(* IEC 61131-3 sources: Codesys_MELSEC_Comm_Sample/src/SLMP_Function, 39 files *)

(* ---- SOCKADDRESS_IN.st ---- *)
TYPE SOCKADDRESS_IN :

STRUCT
    sin_family : INT;
    sin_port   : UINT;
    sin_addr   : UDINT;
    sin_zero   : ARRAY[0..7] OF BYTE;
END_STRUCT
END_TYPE

(* ---- GVL_SlmpConfig.st ---- *)
VAR_GLOBAL CONSTANT
    // LITE preset (active)
    SLMP_MAX_WORD_POINTS : UINT := 120;
    SLMP_MAX_BIT_POINTS : UINT := 960;
    SLMP_MAX_WORD_INDEX : UINT := 119;
    SLMP_MAX_BIT_INDEX : UINT := 959;

    // Buffer sizes for LITE preset (active)
    SLMP_READ_RX_INDEX_MAX : UINT := 511;
    SLMP_WRITE_TX_INDEX_MAX : UINT := 1023;
    SLMP_LAST_RESPONSE_INDEX_MAX : UINT := 63;

    (*
    // FULL preset (commented out)
    SLMP_MAX_WORD_POINTS : UINT := 960;
    SLMP_MAX_BIT_POINTS : UINT := 7168;
    SLMP_MAX_WORD_INDEX : UINT := 959;
    SLMP_MAX_BIT_INDEX : UINT := 7167;

    // Buffer sizes for FULL preset (commented out)
    SLMP_READ_RX_INDEX_MAX : UINT := 4095;
    SLMP_WRITE_TX_INDEX_MAX : UINT := 4095;
    SLMP_LAST_RESPONSE_INDEX_MAX : UINT := 255;
    *)
END_VAR

(* ---- GVL_SlmpDeviceCode.st ---- *)
VAR_GLOBAL CONSTANT
    SLMP_DEV_SM: UINT := 16#0091;
    SLMP_DEV_SD: UINT := 16#00A9;

    SLMP_DEV_X: UINT := 16#009C;
    SLMP_DEV_Y: UINT := 16#009D;

    SLMP_DEV_M: UINT := 16#0090;
    SLMP_DEV_L: UINT := 16#0092;

    SLMP_DEV_F: UINT := 16#0093;
    SLMP_DEV_V: UINT := 16#0094;

    SLMP_DEV_B: UINT := 16#00A0;
    SLMP_DEV_D: UINT := 16#00A8;
    SLMP_DEV_W: UINT := 16#00B4;

    SLMP_DEV_TS: UINT := 16#00C1;
    SLMP_DEV_TC: UINT := 16#00C0;
    SLMP_DEV_TN: UINT := 16#00C2;

    SLMP_DEV_LTS: UINT := 16#0051;
    SLMP_DEV_LTC: UINT := 16#0050;
    SLMP_DEV_LTN: UINT := 16#0052;

    SLMP_DEV_STS: UINT := 16#00C7;
    SLMP_DEV_STC: UINT := 16#00C6;
    SLMP_DEV_STN: UINT := 16#00C8;

    SLMP_DEV_LSTS: UINT := 16#0059;
    SLMP_DEV_LSTC: UINT := 16#0058;
    SLMP_DEV_LSTN: UINT := 16#005A;

    SLMP_DEV_CS: UINT := 16#00C4;
    SLMP_DEV_CC: UINT := 16#00C3;
    SLMP_DEV_CN: UINT := 16#00C5;

    SLMP_DEV_LCS: UINT := 16#0055;
    SLMP_DEV_LCC: UINT := 16#0054;
    SLMP_DEV_LCN: UINT := 16#0056;

    SLMP_DEV_SB: UINT := 16#00A1;
    SLMP_DEV_SW: UINT := 16#00B5;

    SLMP_DEV_S: UINT := 16#0098;

    SLMP_DEV_DX: UINT := 16#00A2;
    SLMP_DEV_DY: UINT := 16#00A3;

    SLMP_DEV_Z: UINT := 16#00CC;
    SLMP_DEV_LZ: UINT := 16#0062;

    SLMP_DEV_R: UINT := 16#00AF;
    SLMP_DEV_ZR: UINT := 16#00B0;

    SLMP_DEV_RD: UINT := 16#002C;
END_VAR

(* ---- GVL_SlmpRuntime.st ---- *)
VAR_GLOBAL
    g_uiSlmpSerialCounter : UINT := 0;
    g_udServiceInstanceCounter : UDINT := 0;
    g_aLockOwner : ARRAY[0..7] OF UDINT := [0,0,0,0,0,0,0,0];
    g_aLockIp : ARRAY[0..7] OF STRING := ['','','','','','','',''];
    g_aLockPort : ARRAY[0..7] OF UINT := [0,0,0,0,0,0,0,0];
    g_aLockUseUdp : ARRAY[0..7] OF BOOL := [FALSE,FALSE,FALSE,FALSE,FALSE,FALSE,FALSE,FALSE];

    g_aSockHandle : ARRAY[0..7] OF RTS_IEC_HANDLE := [
        RTS_INVALID_HANDLE, RTS_INVALID_HANDLE, RTS_INVALID_HANDLE, RTS_INVALID_HANDLE,
        RTS_INVALID_HANDLE, RTS_INVALID_HANDLE, RTS_INVALID_HANDLE, RTS_INVALID_HANDLE
    ];
    g_aSockConnected : ARRAY[0..7] OF BOOL := [FALSE,FALSE,FALSE,FALSE,FALSE,FALSE,FALSE,FALSE];
    g_aSockIp : ARRAY[0..7] OF STRING := ['','','','','','','',''];
    g_aSockPort : ARRAY[0..7] OF UINT := [0,0,0,0,0,0,0,0];
    g_aSockUseUdp : ARRAY[0..7] OF BOOL := [FALSE,FALSE,FALSE,FALSE,FALSE,FALSE,FALSE,FALSE];

    g_aLastTx : ARRAY[0..SLMP_WRITE_TX_INDEX_MAX] OF BYTE := [0];
    g_uiLastTxLen : UINT := 0;
    g_iLastTxSockSlot : INT := -1;
END_VAR

(* ---- GVL_SlmpSubCommand.st ---- *)
VAR_GLOBAL CONSTANT
    SLMP_SUB_WORD  : UINT := 16#0000;
    SLMP_SUB_BIT   : UINT := 16#0001;
    SLMP_SUB_WORD2 : UINT := 16#0002;
    SLMP_SUB_BIT2  : UINT := 16#0003;
END_VAR

(* ---- GVL_SlmpSubCommandByDevice.st ---- *)
VAR_GLOBAL CONSTANT
    SLMP_SUB_DEF_SM   : UINT := SLMP_SUB_BIT;
    SLMP_SUB_DEF_SD   : UINT := SLMP_SUB_WORD;

    SLMP_SUB_DEF_X    : UINT := SLMP_SUB_BIT;
    SLMP_SUB_DEF_Y    : UINT := SLMP_SUB_BIT;
    SLMP_SUB_DEF_M    : UINT := SLMP_SUB_BIT;
    SLMP_SUB_DEF_L    : UINT := SLMP_SUB_BIT;
    SLMP_SUB_DEF_F    : UINT := SLMP_SUB_BIT;
    SLMP_SUB_DEF_V    : UINT := SLMP_SUB_BIT;
    SLMP_SUB_DEF_B    : UINT := SLMP_SUB_BIT;

    SLMP_SUB_DEF_D    : UINT := SLMP_SUB_WORD;
    SLMP_SUB_DEF_W    : UINT := SLMP_SUB_WORD;

    SLMP_SUB_DEF_TS   : UINT := SLMP_SUB_BIT;
    SLMP_SUB_DEF_TC   : UINT := SLMP_SUB_BIT;
    SLMP_SUB_DEF_TN   : UINT := SLMP_SUB_WORD;

    SLMP_SUB_DEF_LTS  : UINT := SLMP_SUB_BIT2;
    SLMP_SUB_DEF_LTC  : UINT := SLMP_SUB_BIT2;
    SLMP_SUB_DEF_LTN  : UINT := SLMP_SUB_WORD2;

    SLMP_SUB_DEF_STS  : UINT := SLMP_SUB_BIT;
    SLMP_SUB_DEF_STC  : UINT := SLMP_SUB_BIT;
    SLMP_SUB_DEF_STN  : UINT := SLMP_SUB_WORD;

    SLMP_SUB_DEF_LSTS : UINT := SLMP_SUB_BIT2;
    SLMP_SUB_DEF_LSTC : UINT := SLMP_SUB_BIT2;
    SLMP_SUB_DEF_LSTN : UINT := SLMP_SUB_WORD2;

    SLMP_SUB_DEF_CS   : UINT := SLMP_SUB_BIT;
    SLMP_SUB_DEF_CC   : UINT := SLMP_SUB_BIT;
    SLMP_SUB_DEF_CN   : UINT := SLMP_SUB_WORD;

    SLMP_SUB_DEF_LCS  : UINT := SLMP_SUB_BIT2;
    SLMP_SUB_DEF_LCC  : UINT := SLMP_SUB_BIT2;
    SLMP_SUB_DEF_LCN  : UINT := SLMP_SUB_WORD;

    SLMP_SUB_DEF_SB   : UINT := SLMP_SUB_BIT;
    SLMP_SUB_DEF_SW   : UINT := SLMP_SUB_WORD;

    SLMP_SUB_DEF_S    : UINT := SLMP_SUB_BIT;

    SLMP_SUB_DEF_DX   : UINT := SLMP_SUB_BIT;
    SLMP_SUB_DEF_DY   : UINT := SLMP_SUB_BIT;

    SLMP_SUB_DEF_Z    : UINT := SLMP_SUB_WORD;
    SLMP_SUB_DEF_LZ   : UINT := SLMP_SUB_WORD2;

    SLMP_SUB_DEF_R    : UINT := SLMP_SUB_WORD;
    SLMP_SUB_DEF_ZR   : UINT := SLMP_SUB_WORD;

    SLMP_SUB_DEF_RD   : UINT := SLMP_SUB_WORD2;

END_VAR

(* ---- F_SlmpAutoSubCommand.st ---- *)
FUNCTION F_SlmpAutoSubCommand : UINT
VAR_INPUT
    uiDeviceCode : UINT;
END_VAR

// === IMPLEMENTATION ===
CASE uiDeviceCode OF
    SLMP_DEV_D: F_SlmpAutoSubCommand := SLMP_SUB_DEF_D;
    SLMP_DEV_M: F_SlmpAutoSubCommand := SLMP_SUB_DEF_M;
    SLMP_DEV_X: F_SlmpAutoSubCommand := SLMP_SUB_DEF_X;
    SLMP_DEV_Y: F_SlmpAutoSubCommand := SLMP_SUB_DEF_Y;
    SLMP_DEV_L: F_SlmpAutoSubCommand := SLMP_SUB_DEF_L;
    SLMP_DEV_SM: F_SlmpAutoSubCommand := SLMP_SUB_DEF_SM;
    SLMP_DEV_SD: F_SlmpAutoSubCommand := SLMP_SUB_DEF_SD;
    SLMP_DEV_F: F_SlmpAutoSubCommand := SLMP_SUB_DEF_F;
    SLMP_DEV_V: F_SlmpAutoSubCommand := SLMP_SUB_DEF_V;
    SLMP_DEV_R: F_SlmpAutoSubCommand := SLMP_SUB_DEF_R;
    SLMP_DEV_W: F_SlmpAutoSubCommand := SLMP_SUB_DEF_W;
    SLMP_DEV_B: F_SlmpAutoSubCommand := SLMP_SUB_DEF_B;
    SLMP_DEV_TS: F_SlmpAutoSubCommand := SLMP_SUB_DEF_TS;
    SLMP_DEV_TC: F_SlmpAutoSubCommand := SLMP_SUB_DEF_TC;
    SLMP_DEV_TN: F_SlmpAutoSubCommand := SLMP_SUB_DEF_TN;
    SLMP_DEV_LTS: F_SlmpAutoSubCommand := SLMP_SUB_DEF_LTS;
    SLMP_DEV_LTC: F_SlmpAutoSubCommand := SLMP_SUB_DEF_LTC;
    SLMP_DEV_LTN: F_SlmpAutoSubCommand := SLMP_SUB_DEF_LTN;
    SLMP_DEV_STS: F_SlmpAutoSubCommand := SLMP_SUB_DEF_STS;
    SLMP_DEV_STC: F_SlmpAutoSubCommand := SLMP_SUB_DEF_STC;
    SLMP_DEV_STN: F_SlmpAutoSubCommand := SLMP_SUB_DEF_STN;
    SLMP_DEV_LSTS: F_SlmpAutoSubCommand := SLMP_SUB_DEF_LSTS;
    SLMP_DEV_LSTC: F_SlmpAutoSubCommand := SLMP_SUB_DEF_LSTC;
    SLMP_DEV_LSTN: F_SlmpAutoSubCommand := SLMP_SUB_DEF_LSTN;
    SLMP_DEV_CS: F_SlmpAutoSubCommand := SLMP_SUB_DEF_CS;
    SLMP_DEV_CC: F_SlmpAutoSubCommand := SLMP_SUB_DEF_CC;
    SLMP_DEV_CN: F_SlmpAutoSubCommand := SLMP_SUB_DEF_CN;
    SLMP_DEV_LCS: F_SlmpAutoSubCommand := SLMP_SUB_DEF_LCS;
    SLMP_DEV_LCC: F_SlmpAutoSubCommand := SLMP_SUB_DEF_LCC;
    SLMP_DEV_LCN: F_SlmpAutoSubCommand := SLMP_SUB_DEF_LCN;
    SLMP_DEV_SB: F_SlmpAutoSubCommand := SLMP_SUB_DEF_SB;
    SLMP_DEV_SW: F_SlmpAutoSubCommand := SLMP_SUB_DEF_SW;
    SLMP_DEV_ZR: F_SlmpAutoSubCommand := SLMP_SUB_DEF_ZR;
    SLMP_DEV_DX: F_SlmpAutoSubCommand := SLMP_SUB_DEF_DX;
    SLMP_DEV_DY: F_SlmpAutoSubCommand := SLMP_SUB_DEF_DY;
    SLMP_DEV_S: F_SlmpAutoSubCommand := SLMP_SUB_DEF_S;
    SLMP_DEV_Z: F_SlmpAutoSubCommand := SLMP_SUB_DEF_Z;
    SLMP_DEV_LZ: F_SlmpAutoSubCommand := SLMP_SUB_DEF_LZ;
    SLMP_DEV_RD: F_SlmpAutoSubCommand := SLMP_SUB_DEF_RD;
ELSE
    F_SlmpAutoSubCommand := SLMP_SUB_WORD;
END_CASE;

(* ---- F_SlmpClampPoints.st ---- *)
FUNCTION F_SlmpClampPoints : UINT
VAR_INPUT
    uiPoints : UINT;
    xBitMode : BOOL;
END_VAR

// === IMPLEMENTATION ===
IF uiPoints = 0 THEN
    F_SlmpClampPoints := 0;
ELSIF xBitMode THEN
    IF uiPoints > SLMP_MAX_BIT_POINTS THEN
        F_SlmpClampPoints := SLMP_MAX_BIT_POINTS;
    ELSE
        F_SlmpClampPoints := uiPoints;
    END_IF;
ELSE
    IF uiPoints > SLMP_MAX_WORD_POINTS THEN
        F_SlmpClampPoints := SLMP_MAX_WORD_POINTS;
    ELSE
        F_SlmpClampPoints := uiPoints;
    END_IF;
END_IF;

(* ---- F_SlmpEndCodeText.st ---- *)
FUNCTION F_SlmpEndCodeText : STRING
VAR_INPUT
    uiEndCode : UINT;
END_VAR

// === IMPLEMENTATION ===
CASE uiEndCode OF
    16#0000: F_SlmpEndCodeText := 'OK';
    16#0050: F_SlmpEndCodeText := 'OUT_OF_RANGE';
    16#C051: F_SlmpEndCodeText := 'POINTS_OR_HEAD_DEVICE_ERROR';
    16#C052: F_SlmpEndCodeText := 'COMMAND_NOT_SUPPORTED';
    16#C053: F_SlmpEndCodeText := 'SUBCOMMAND_NOT_SUPPORTED';
    16#C054: F_SlmpEndCodeText := 'DATA_FORMAT_ERROR';
    16#C055: F_SlmpEndCodeText := 'WRITE_PROTECTED';
    16#C056: F_SlmpEndCodeText := 'CPU_BUSY';
    16#C061: F_SlmpEndCodeText := 'REQUEST_DATA_LENGTH_ERROR';
    16#CE10: F_SlmpEndCodeText := 'NETWORK_PARAMETER_ERROR';
    16#CE11: F_SlmpEndCodeText := 'DESTINATION_PARAMETER_ERROR';
ELSE
    F_SlmpEndCodeText := 'UNKNOWN_END_CODE';
END_CASE;

(* ---- F_SlmpIsBitSubCommand.st ---- *)
FUNCTION F_SlmpIsBitSubCommand : BOOL
VAR_INPUT
    uiSubCommand : UINT;
END_VAR

// === IMPLEMENTATION ===
F_SlmpIsBitSubCommand := (uiSubCommand = SLMP_SUB_BIT) OR (uiSubCommand = SLMP_SUB_BIT2);

(* ---- F_SlmpNextSerialNo.st ---- *)
FUNCTION F_SlmpNextSerialNo : UINT
VAR_INPUT
    uiSeed : UINT := 1;
END_VAR

// === IMPLEMENTATION ===
IF g_uiSlmpSerialCounter = 0 THEN
    IF uiSeed = 0 THEN
        g_uiSlmpSerialCounter := 1;
    ELSE
        g_uiSlmpSerialCounter := uiSeed;
    END_IF;
ELSE
    g_uiSlmpSerialCounter := g_uiSlmpSerialCounter + 1;
    IF g_uiSlmpSerialCounter = 0 THEN
        g_uiSlmpSerialCounter := 1;
    END_IF;
END_IF;

F_SlmpNextSerialNo := g_uiSlmpSerialCounter;

(* ---- F_SlmpResolveSubCommand.st ---- *)
FUNCTION F_SlmpResolveSubCommand : UINT
VAR_INPUT
    uiDeviceCode    : UINT;
    xAutoSubCommand : BOOL;
    uiSubCommand    : UINT;
END_VAR

// === IMPLEMENTATION ===
IF xAutoSubCommand THEN
    F_SlmpResolveSubCommand := F_SlmpAutoSubCommand(uiDeviceCode := uiDeviceCode);
ELSE
    F_SlmpResolveSubCommand := uiSubCommand;
END_IF;

(* ---- FB_SlmpCloseConnection.st ---- *)
FUNCTION_BLOCK FB_SlmpCloseConnection
VAR_INPUT
    xExecute : BOOL;
END_VAR
VAR_OUTPUT
    xDone    : BOOL;
END_VAR
VAR
    xExecPrev : BOOL := FALSE;
    iSlot     : INT := 0;
END_VAR

// === IMPLEMENTATION ===
xDone := FALSE;

IF xExecute AND (NOT xExecPrev) THEN
    FOR iSlot := 0 TO 7 DO
        IF GVL_SlmpRuntime.g_aSockHandle[iSlot] <> RTS_INVALID_HANDLE THEN
            SysSockClose(GVL_SlmpRuntime.g_aSockHandle[iSlot]);
            GVL_SlmpRuntime.g_aSockHandle[iSlot] := RTS_INVALID_HANDLE;
        END_IF;
        GVL_SlmpRuntime.g_aSockConnected[iSlot] := FALSE;
        GVL_SlmpRuntime.g_aSockIp[iSlot] := '';
        GVL_SlmpRuntime.g_aSockPort[iSlot] := 0;
        GVL_SlmpRuntime.g_aSockUseUdp[iSlot] := FALSE;

        GVL_SlmpRuntime.g_aLockOwner[iSlot] := 0;
        GVL_SlmpRuntime.g_aLockIp[iSlot] := '';
        GVL_SlmpRuntime.g_aLockPort[iSlot] := 0;
        GVL_SlmpRuntime.g_aLockUseUdp[iSlot] := FALSE;
    END_FOR;
    xDone := TRUE;
END_IF;

xExecPrev := xExecute;

(* ---- FB_SlmpCore.st ---- *)
FUNCTION_BLOCK FB_SlmpCore
VAR_OUTPUT
    diLastError : DINT;
END_VAR
VAR
    iSockSlot      : INT := -1;
    res            : RTS_IEC_RESULT := 0;
    sa             : SOCKADDRESS_IN;
    ipAddr         : UDINT := 0;
    liRet          : LINT := 0;
END_VAR

(* ---- FB_SlmpReadBitDevice.st ---- *)
FUNCTION_BLOCK FB_SlmpReadBitDevice
VAR_INPUT
    xExecute         : BOOL;
    sIp              : STRING;
    uiPort           : UINT;
    udiHeadDevNo     : UDINT := 100;
    uiDeviceCode     : UINT := 16#0090; // M
    xAutoSubCommand  : BOOL := TRUE;
    uiSubCommand     : UINT := 16#0001;
    uiPoints         : UINT := 1;
    tTimeout         : TIME := T#2S;
    uiRetryMax       : UINT := 2;
    tReconnectDelay  : TIME := T#500MS;
    xUse4E           : BOOL := FALSE;
    xUseUdp          : BOOL := FALSE;
    uiSerialNo       : UINT := 0;
END_VAR
VAR_OUTPUT
    xBusy            : BOOL;
    xDone            : BOOL;
    xError           : BOOL;
    diError          : DINT;
    uiRetryCount     : UINT;
    uiReadBits       : UINT;
    uiValue0         : UINT;
    aBits            : ARRAY[0..SLMP_MAX_BIT_INDEX] OF BOOL;
    aLastResponse    : ARRAY[0..SLMP_LAST_RESPONSE_INDEX_MAX] OF BYTE;
    uiLastResponseLen: UINT;
    uiLastEndCode    : UINT;
END_VAR
VAR
    step             : INT := 0;
    xExecPrev        : BOOL := FALSE;

    fbCore           : FB_SlmpCore;

    tx               : ARRAY[0..31] OF BYTE;
    rx               : ARRAY[0..SLMP_READ_RX_INDEX_MAX] OF BYTE;
    txLen            : LINT := 0;
    rxLen            : LINT := 0;
    lenReq           : UINT := 0;
    endCode          : UINT := 0;

    uiPointsReq      : UINT := 0;
    uiPointsEff      : UINT := 0;
    uiSubCmdEff      : UINT := 0;
    iDataStart       : DINT := 11;
    iEndCodeStart    : DINT := 9;
    iNeedRxLen       : LINT := 0;
    uiRxSerialNo     : UINT := 0;
    uiCopyLen        : UINT := 0;
    iByteOffset      : DINT := 0;
    byData           : BYTE := 0;
    idx              : UINT := 0;

    xStateTimeout    : BOOL := FALSE;
    xRetryTiming     : BOOL := FALSE;
    fbTimeout        : TON;
    fbReconnect      : TON;
END_VAR

// === IMPLEMENTATION ===
IF (xExecute AND NOT xExecPrev) THEN
    xBusy := TRUE;
    xDone := FALSE;
    xError := FALSE;
    diError := 0;
    uiRetryCount := 0;
    uiReadBits := 0;
    uiValue0 := 0;
    uiLastResponseLen := 0;
    uiLastEndCode := 0;
    FOR idx := 0 TO SLMP_MAX_BIT_INDEX DO
        aBits[idx] := FALSE;
    END_FOR;
    FOR idx := 0 TO SLMP_LAST_RESPONSE_INDEX_MAX DO
        aLastResponse[idx] := 0;
    END_FOR;
    step := 10;
END_IF;
xExecPrev := xExecute;

xStateTimeout := (step = 20) OR (step = 40) OR (step = 50);
fbTimeout(IN := xStateTimeout, PT := tTimeout);
fbReconnect(IN := xRetryTiming, PT := tReconnectDelay);

IF (step <> 0) AND (step <> 80) AND fbTimeout.Q THEN
    diError := -1010;
    xError := TRUE;
    step := 90;
END_IF;

CASE step OF
    0:
        xRetryTiming := FALSE;

    10:
        uiSubCmdEff := F_SlmpResolveSubCommand(
            uiDeviceCode := uiDeviceCode,
            xAutoSubCommand := xAutoSubCommand,
            uiSubCommand := uiSubCommand
        );

        uiPointsReq := uiPoints;
        IF uiPointsReq = 0 THEN
            diError := -1000;
            xError := TRUE;
            xBusy := FALSE;
            step := 0;
        ELSE
            uiPointsEff := F_SlmpClampPoints(uiPoints := uiPointsReq, xBitMode := TRUE);
        END_IF;

        IF NOT xError THEN
            step := 20;
        END_IF;

    20:
        IF fbCore.OpenAndConnect(sIp := sIp, uiPort := uiPort, xUseUdp := xUseUdp) THEN
            step := 30;
        ELSE
            CASE fbCore.diLastError OF
                -1: diError := -1001;
                -2: diError := -1005;
                -3: diError := -1002;
            ELSE
                diError := -1002;
            END_CASE;
            xError := TRUE;
            step := 90;
        END_IF;

    30:
        lenReq := 12;
        IF xUse4E THEN
            iDataStart := 15;
            iEndCodeStart := 13;
            tx[0] := 16#54; tx[1] := 16#00;
            tx[2] := TO_BYTE(uiSerialNo AND 16#00FF);
            tx[3] := TO_BYTE(SHR(uiSerialNo, 8) AND 16#00FF);
            tx[4] := 16#00; tx[5] := 16#00;
            tx[6] := 16#00;
            tx[7] := 16#FF;
            tx[8] := 16#FF; tx[9] := 16#03;
            tx[10] := 16#00;
            tx[11] := TO_BYTE(lenReq AND 16#00FF);
            tx[12] := TO_BYTE(SHR(lenReq, 8) AND 16#00FF);
            tx[13] := 16#10; tx[14] := 16#00;
            tx[15] := 16#01; tx[16] := 16#04;
            tx[17] := TO_BYTE(uiSubCmdEff AND 16#00FF);
            tx[18] := TO_BYTE(SHR(uiSubCmdEff, 8) AND 16#00FF);
            tx[19] := TO_BYTE(udiHeadDevNo AND 16#000000FF);
            tx[20] := TO_BYTE(SHR(udiHeadDevNo, 8) AND 16#000000FF);
            tx[21] := TO_BYTE(SHR(udiHeadDevNo, 16) AND 16#000000FF);
            tx[22] := TO_BYTE(uiDeviceCode AND 16#00FF);
            tx[23] := TO_BYTE(uiPointsEff AND 16#00FF);
            tx[24] := TO_BYTE(SHR(uiPointsEff, 8) AND 16#00FF);
            txLen := 25;
        ELSE
            iDataStart := 11;
            iEndCodeStart := 9;
            tx[0] := 16#50; tx[1] := 16#00;
            tx[2] := 16#00;
            tx[3] := 16#FF;
            tx[4] := 16#FF; tx[5] := 16#03;
            tx[6] := 16#00;
            tx[7] := TO_BYTE(lenReq AND 16#00FF);
            tx[8] := TO_BYTE(SHR(lenReq, 8) AND 16#00FF);
            tx[9] := 16#10; tx[10] := 16#00;
            tx[11] := 16#01; tx[12] := 16#04;
            tx[13] := TO_BYTE(uiSubCmdEff AND 16#00FF);
            tx[14] := TO_BYTE(SHR(uiSubCmdEff, 8) AND 16#00FF);
            tx[15] := TO_BYTE(udiHeadDevNo AND 16#000000FF);
            tx[16] := TO_BYTE(SHR(udiHeadDevNo, 8) AND 16#000000FF);
            tx[17] := TO_BYTE(SHR(udiHeadDevNo, 16) AND 16#000000FF);
            tx[18] := TO_BYTE(uiDeviceCode AND 16#00FF);
            tx[19] := TO_BYTE(uiPointsEff AND 16#00FF);
            tx[20] := TO_BYTE(SHR(uiPointsEff, 8) AND 16#00FF);
            txLen := 21;
        END_IF;
        step := 40;

    40:
        IF NOT fbCore.SendBytes(pData := ADR(tx[0]), liLen := txLen) THEN
            diError := -1003;
            xError := TRUE;
            step := 90;
        ELSE
            step := 50;
        END_IF;

    50:
        rxLen := fbCore.RecvBytes(pData := ADR(rx[0]), liMaxLen := SIZEOF(rx));
        IF rxLen > 0 THEN
            uiCopyLen := 0;
            IF rxLen > TO_LINT(SLMP_LAST_RESPONSE_INDEX_MAX + 1) THEN
                uiCopyLen := SLMP_LAST_RESPONSE_INDEX_MAX + 1;
            ELSE
                uiCopyLen := TO_UINT(rxLen);
            END_IF;
            uiLastResponseLen := uiCopyLen;
            IF uiCopyLen > 0 THEN
                FOR idx := 0 TO (uiCopyLen - 1) DO
                    aLastResponse[idx] := rx[idx];
                END_FOR;
            END_IF;

            iNeedRxLen := iDataStart + TO_LINT((uiPointsEff + 1) / 2);
            IF rxLen < iNeedRxLen THEN
                diError := -1004;
                xError := TRUE;
                step := 90;
            ELSE
                IF xUse4E THEN
                    uiRxSerialNo := TO_UINT(rx[2]) OR SHL(TO_UINT(rx[3]), 8);
                    IF uiRxSerialNo <> uiSerialNo THEN
                        // Drop stale frame and keep waiting until timeout.
                        rxLen := 0;
                        uiLastResponseLen := 0;
                    END_IF;
                END_IF;
            END_IF;
            IF (NOT xError) AND (rxLen > 0) THEN
                endCode := TO_UINT(rx[iEndCodeStart]) OR SHL(TO_UINT(rx[iEndCodeStart + 1]), 8);
                uiLastEndCode := endCode;
                IF endCode <> 0 THEN
                    diError := TO_DINT(endCode);
                    xError := TRUE;
                    step := 90;
                ELSE
                    FOR idx := 0 TO (uiPointsEff - 1) DO
                        iByteOffset := iDataStart + TO_DINT(idx / 2);
                        byData := rx[iByteOffset];
                        IF (idx MOD 2) = 0 THEN
                            aBits[idx] := (byData AND 16#F0) <> 0;
                        ELSE
                            aBits[idx] := (byData AND 16#0F) <> 0;
                        END_IF;
                    END_FOR;
                    uiReadBits := uiPointsEff;
                    IF uiPointsEff > 0 THEN
                        IF aBits[0] THEN
                            uiValue0 := 1;
                        ELSE
                            uiValue0 := 0;
                        END_IF;
                    END_IF;
                    xDone := TRUE;
                    xBusy := FALSE;
                    step := 90;
                END_IF;
            END_IF;
        END_IF;

    80:
        xRetryTiming := TRUE;
        IF fbReconnect.Q THEN
            xRetryTiming := FALSE;
            step := 10;
        END_IF;

    90:
        IF xError THEN
            fbCore.CloseSocket();
        END_IF;

        IF xError AND (uiRetryCount < uiRetryMax) THEN
            uiRetryCount := uiRetryCount + 1;
            xError := FALSE;
            step := 80;
        ELSE
            xBusy := FALSE;
            step := 0;
        END_IF;
END_CASE;

(* ---- FB_SlmpReadBitService.st ---- *)
FUNCTION_BLOCK FB_SlmpReadBitService
VAR_INPUT
    xExecute        : BOOL;
    sIp             : STRING;
    uiPort          : UINT;
    udiHeadDevNo    : UDINT;
    uiDeviceCode    : UINT;
    uiPoints        : UINT;
    tTimeout        : TIME := T#2S;
    uiRetryMax      : UINT := 2;
    tReconnectDelay : TIME := T#500MS;
    xUse4E          : BOOL := FALSE;
    xUseUdp         : BOOL := FALSE;
    uiSerialNo      : UINT := 1;
END_VAR
VAR_OUTPUT
    xBusy           : BOOL;
    xDone           : BOOL;
    xError          : BOOL;
    diError         : DINT;
    uiRetryCount    : UINT;
    uiReadBits      : UINT;
    uiValue0        : UINT;
    aReadBits       : ARRAY[0..SLMP_MAX_BIT_INDEX] OF BOOL;
    aLastResponse   : ARRAY[0..SLMP_LAST_RESPONSE_INDEX_MAX] OF BYTE;
    uiLastResponseLen : UINT;
    uiLastEndCode   : UINT;
END_VAR
VAR
    fbReadBit       : FB_SlmpReadBitDevice;
    udInstanceId    : UDINT := 0;

    xExecPrev       : BOOL := FALSE;
    xPending        : BOOL := FALSE;
    xActive         : BOOL := FALSE;
    xExecPulse      : BOOL := FALSE;
    iLockIdx        : INT := -1;

    udiHeadLatched  : UDINT := 0;
    uiDeviceLatched : UINT := 0;
    uiPointsLatched : UINT := 0;
    uiSerialActive  : UINT := 0;

    idx             : UINT;
    uiSerialEff     : UINT;
    iSlot           : INT;
    iFreeSlot       : INT;
    xLocked         : BOOL;
END_VAR

// === IMPLEMENTATION ===
IF udInstanceId = 0 THEN
    GVL_SlmpRuntime.g_udServiceInstanceCounter := GVL_SlmpRuntime.g_udServiceInstanceCounter + 1;
    udInstanceId := GVL_SlmpRuntime.g_udServiceInstanceCounter;
    IF udInstanceId = 0 THEN
        udInstanceId := 1;
    END_IF;
END_IF;

IF xExecute AND (NOT xExecPrev) THEN
    IF (NOT xPending) AND (NOT xActive) THEN
        udiHeadLatched := udiHeadDevNo;
        uiDeviceLatched := uiDeviceCode;
        uiPointsLatched := uiPoints;
        xDone := FALSE;
        xError := FALSE;
        diError := 0;
        uiRetryCount := 0;
        xPending := TRUE;
    END_IF;
END_IF;
xExecPrev := xExecute;

xExecPulse := FALSE;
IF xPending AND (NOT xActive) THEN
    xLocked := FALSE;
    iFreeSlot := -1;
    FOR iSlot := 0 TO 7 DO
        IF (GVL_SlmpRuntime.g_aLockOwner[iSlot] <> 0) AND
           (GVL_SlmpRuntime.g_aLockIp[iSlot] = sIp) AND
           (GVL_SlmpRuntime.g_aLockPort[iSlot] = uiPort) AND
           (GVL_SlmpRuntime.g_aLockUseUdp[iSlot] = xUseUdp) THEN
            xLocked := TRUE;
            EXIT;
        END_IF;
        IF (iFreeSlot < 0) AND (GVL_SlmpRuntime.g_aLockOwner[iSlot] = 0) THEN
            iFreeSlot := iSlot;
        END_IF;
    END_FOR;

    IF (NOT xLocked) AND (iFreeSlot >= 0) THEN
        GVL_SlmpRuntime.g_aLockOwner[iFreeSlot] := udInstanceId;
        GVL_SlmpRuntime.g_aLockIp[iFreeSlot] := sIp;
        GVL_SlmpRuntime.g_aLockPort[iFreeSlot] := uiPort;
        GVL_SlmpRuntime.g_aLockUseUdp[iFreeSlot] := xUseUdp;
        iLockIdx := iFreeSlot;

        xActive := TRUE;
        xExecPulse := TRUE;
        IF xUse4E THEN
            uiSerialActive := F_SlmpNextSerialNo(uiSeed := uiSerialNo);
        END_IF;
    END_IF;
END_IF;

IF xActive THEN
    IF xUse4E THEN
        uiSerialEff := uiSerialActive;
        IF uiSerialEff = 0 THEN
            uiSerialEff := 1;
        END_IF;
    ELSE
        uiSerialEff := uiSerialNo;
    END_IF;

    fbReadBit(
        xExecute := xExecPulse,
        sIp := sIp,
        uiPort := uiPort,
        udiHeadDevNo := udiHeadLatched,
        uiDeviceCode := uiDeviceLatched,
        xAutoSubCommand := TRUE,
        uiSubCommand := 0,
        uiPoints := uiPointsLatched,
        tTimeout := tTimeout,
        uiRetryMax := uiRetryMax,
        tReconnectDelay := tReconnectDelay,
        xUse4E := xUse4E,
        xUseUdp := xUseUdp,
        uiSerialNo := uiSerialEff
    );
ELSE
    xBusy := xPending;
    IF NOT xExecute THEN
        xDone := FALSE;
        xError := FALSE;
        diError := 0;
        uiRetryCount := 0;
    END_IF;
    RETURN;
END_IF;

xBusy := fbReadBit.xBusy;
xDone := fbReadBit.xDone;
xError := fbReadBit.xError;
diError := fbReadBit.diError;
uiRetryCount := fbReadBit.uiRetryCount;

IF fbReadBit.xDone THEN
    uiReadBits := fbReadBit.uiReadBits;
    uiValue0 := fbReadBit.uiValue0;
    FOR idx := 0 TO SLMP_MAX_BIT_INDEX DO
        aReadBits[idx] := fbReadBit.aBits[idx];
    END_FOR;
    FOR idx := 0 TO SLMP_LAST_RESPONSE_INDEX_MAX DO
        aLastResponse[idx] := fbReadBit.aLastResponse[idx];
    END_FOR;
    uiLastResponseLen := fbReadBit.uiLastResponseLen;
    uiLastEndCode := fbReadBit.uiLastEndCode;
END_IF;

IF fbReadBit.xDone OR fbReadBit.xError THEN
    xPending := FALSE;
    xActive := FALSE;
    IF iLockIdx >= 0 THEN
        GVL_SlmpRuntime.g_aLockOwner[iLockIdx] := 0;
        GVL_SlmpRuntime.g_aLockIp[iLockIdx] := '';
        GVL_SlmpRuntime.g_aLockPort[iLockIdx] := 0;
        GVL_SlmpRuntime.g_aLockUseUdp[iLockIdx] := FALSE;
        iLockIdx := -1;
    END_IF;
END_IF;

(* ---- FB_SlmpReadDevice.st ---- *)
FUNCTION_BLOCK FB_SlmpReadDevice
VAR_INPUT
    xExecute         : BOOL;
    sIp              : STRING;
    uiPort           : UINT;
    udiHeadDevNo     : UDINT := 100;
    uiDeviceCode     : UINT := 16#00A8; // D
    xAutoSubCommand  : BOOL := TRUE;
    uiSubCommand     : UINT := 16#0000; // 0000: word, 0001: bit
    uiPoints         : UINT := 1;
    tTimeout         : TIME := T#2S;
    uiRetryMax       : UINT := 2;
    tReconnectDelay  : TIME := T#500MS;
    xUse4E           : BOOL := FALSE;
    uiSerialNo       : UINT := 0;
END_VAR
VAR_OUTPUT
    xBusy            : BOOL;
    xDone            : BOOL;
    xError           : BOOL;
    diError          : DINT;
    uiRetryCount     : UINT;
    uiReadWords      : UINT;
    uiReadBits       : UINT;
    uiValue0         : UINT;
    aValues          : ARRAY[0..SLMP_MAX_WORD_INDEX] OF UINT;
    aBits            : ARRAY[0..SLMP_MAX_BIT_INDEX] OF BOOL;
    aLastResponse    : ARRAY[0..SLMP_LAST_RESPONSE_INDEX_MAX] OF BYTE;
    uiLastResponseLen: UINT;
    uiLastEndCode    : UINT;
END_VAR
VAR
    step             : INT := 0;
    xExecPrev        : BOOL := FALSE;

    fbCore           : FB_SlmpCore;

    tx               : ARRAY[0..31] OF BYTE;
    rx               : ARRAY[0..SLMP_READ_RX_INDEX_MAX] OF BYTE;
    txLen            : LINT := 0;
    rxLen            : LINT := 0;
    lenReq           : UINT := 0;
    endCode          : UINT := 0;

    uiPointsReq      : UINT := 0;
    uiPointsEff      : UINT := 0;
    uiSubCmdEff      : UINT := 0;
    iDataStart       : DINT := 11;
    iEndCodeStart    : DINT := 9;
    iNeedRxLen       : LINT := 0;
    uiRxSerialNo     : UINT := 0;
    uiCopyLen        : UINT := 0;
    iByteOffset      : DINT := 0;
    byData           : BYTE := 0;
    idx              : UINT := 0;
    xBitMode         : BOOL := FALSE;

    xStateTimeout    : BOOL := FALSE;
    xRetryTiming     : BOOL := FALSE;
    fbTimeout        : TON;
    fbReconnect      : TON;
END_VAR

// === IMPLEMENTATION ===
IF (xExecute AND NOT xExecPrev) THEN
    xBusy := TRUE;
    xDone := FALSE;
    xError := FALSE;
    diError := 0;
    uiRetryCount := 0;
    uiReadWords := 0;
    uiReadBits := 0;
    uiValue0 := 0;
    uiLastResponseLen := 0;
    uiLastEndCode := 0;
    FOR idx := 0 TO SLMP_MAX_WORD_INDEX DO
        aValues[idx] := 0;
    END_FOR;
    FOR idx := 0 TO SLMP_MAX_BIT_INDEX DO
        aBits[idx] := FALSE;
    END_FOR;
    FOR idx := 0 TO SLMP_LAST_RESPONSE_INDEX_MAX DO
        aLastResponse[idx] := 0;
    END_FOR;
    step := 10;
END_IF;
xExecPrev := xExecute;

xStateTimeout := (step = 20) OR (step = 40) OR (step = 50);
fbTimeout(IN := xStateTimeout, PT := tTimeout);
fbReconnect(IN := xRetryTiming, PT := tReconnectDelay);

IF (step <> 0) AND (step <> 80) AND fbTimeout.Q THEN
    diError := -1010;
    xError := TRUE;
    step := 90;
END_IF;

CASE step OF
    0:
        xRetryTiming := FALSE;

    10:
        uiSubCmdEff := F_SlmpResolveSubCommand(
            uiDeviceCode := uiDeviceCode,
            xAutoSubCommand := xAutoSubCommand,
            uiSubCommand := uiSubCommand
        );
        xBitMode := F_SlmpIsBitSubCommand(uiSubCommand := uiSubCmdEff);

        uiPointsReq := uiPoints;
        IF uiPointsReq = 0 THEN
            diError := -1000;
            xError := TRUE;
            xBusy := FALSE;
            step := 0;
        ELSE
            uiPointsEff := F_SlmpClampPoints(uiPoints := uiPointsReq, xBitMode := xBitMode);
        END_IF;

        IF NOT xError THEN
            step := 20;
        END_IF;

    20:
        IF fbCore.OpenAndConnect(sIp := sIp, uiPort := uiPort) THEN
            step := 30;
        ELSE
            CASE fbCore.diLastError OF
                -1: diError := -1001;
                -2: diError := -1005;
                -3: diError := -1002;
            ELSE
                diError := -1002;
            END_CASE;
            xError := TRUE;
            step := 90;
        END_IF;

    30:
        lenReq := 12;
        IF xUse4E THEN
            iDataStart := 15;
            iEndCodeStart := 13;
            tx[0] := 16#54; tx[1] := 16#00;
            tx[2] := TO_BYTE(uiSerialNo AND 16#00FF);
            tx[3] := TO_BYTE(SHR(uiSerialNo, 8) AND 16#00FF);
            tx[4] := 16#00; tx[5] := 16#00;
            tx[6] := 16#00;
            tx[7] := 16#FF;
            tx[8] := 16#FF; tx[9] := 16#03;
            tx[10] := 16#00;
            tx[11] := TO_BYTE(lenReq AND 16#00FF);
            tx[12] := TO_BYTE(SHR(lenReq, 8) AND 16#00FF);
            tx[13] := 16#10; tx[14] := 16#00;
            tx[15] := 16#01; tx[16] := 16#04;
            tx[17] := TO_BYTE(uiSubCmdEff AND 16#00FF);
            tx[18] := TO_BYTE(SHR(uiSubCmdEff, 8) AND 16#00FF);
            tx[19] := TO_BYTE(udiHeadDevNo AND 16#000000FF);
            tx[20] := TO_BYTE(SHR(udiHeadDevNo, 8) AND 16#000000FF);
            tx[21] := TO_BYTE(SHR(udiHeadDevNo, 16) AND 16#000000FF);
            tx[22] := TO_BYTE(uiDeviceCode AND 16#00FF);
            tx[23] := TO_BYTE(uiPointsEff AND 16#00FF);
            tx[24] := TO_BYTE(SHR(uiPointsEff, 8) AND 16#00FF);
            txLen := 25;
        ELSE
            iDataStart := 11;
            iEndCodeStart := 9;
            tx[0] := 16#50; tx[1] := 16#00;
            tx[2] := 16#00;
            tx[3] := 16#FF;
            tx[4] := 16#FF; tx[5] := 16#03;
            tx[6] := 16#00;
            tx[7] := TO_BYTE(lenReq AND 16#00FF);
            tx[8] := TO_BYTE(SHR(lenReq, 8) AND 16#00FF);
            tx[9] := 16#10; tx[10] := 16#00;
            tx[11] := 16#01; tx[12] := 16#04;
            tx[13] := TO_BYTE(uiSubCmdEff AND 16#00FF);
            tx[14] := TO_BYTE(SHR(uiSubCmdEff, 8) AND 16#00FF);
            tx[15] := TO_BYTE(udiHeadDevNo AND 16#000000FF);
            tx[16] := TO_BYTE(SHR(udiHeadDevNo, 8) AND 16#000000FF);
            tx[17] := TO_BYTE(SHR(udiHeadDevNo, 16) AND 16#000000FF);
            tx[18] := TO_BYTE(uiDeviceCode AND 16#00FF);
            tx[19] := TO_BYTE(uiPointsEff AND 16#00FF);
            tx[20] := TO_BYTE(SHR(uiPointsEff, 8) AND 16#00FF);
            txLen := 21;
        END_IF;
        step := 40;

    40:
        IF NOT fbCore.SendBytes(pData := ADR(tx[0]), liLen := txLen) THEN
            diError := -1003;
            xError := TRUE;
            step := 90;
        ELSE
            step := 50;
        END_IF;

    50:
        rxLen := fbCore.RecvBytes(pData := ADR(rx[0]), liMaxLen := SIZEOF(rx));
        IF rxLen > 0 THEN
            uiCopyLen := 0;
            IF rxLen > TO_LINT(SLMP_LAST_RESPONSE_INDEX_MAX + 1) THEN
                uiCopyLen := SLMP_LAST_RESPONSE_INDEX_MAX + 1;
            ELSE
                uiCopyLen := TO_UINT(rxLen);
            END_IF;
            uiLastResponseLen := uiCopyLen;
            IF uiCopyLen > 0 THEN
                FOR idx := 0 TO (uiCopyLen - 1) DO
                    aLastResponse[idx] := rx[idx];
                END_FOR;
            END_IF;
            iNeedRxLen := CalcNeedRxLen();
            IF rxLen < iNeedRxLen THEN
                diError := -1004;
                xError := TRUE;
                step := 90;
            ELSE
                IF xUse4E THEN
                    uiRxSerialNo := TO_UINT(rx[2]) OR SHL(TO_UINT(rx[3]), 8);
                    IF uiRxSerialNo <> uiSerialNo THEN
                        // Drop stale frame and keep waiting until timeout.
                        rxLen := 0;
                        uiLastResponseLen := 0;
                    END_IF;
                END_IF;
            END_IF;
            IF (NOT xError) AND (rxLen > 0) THEN
                endCode := TO_UINT(rx[iEndCodeStart]) OR SHL(TO_UINT(rx[iEndCodeStart + 1]), 8);
                uiLastEndCode := endCode;
                IF endCode <> 0 THEN
                    diError := TO_DINT(endCode);
                    xError := TRUE;
                    step := 90;
                ELSE
                    DecodeReadData();
                    xDone := TRUE;
                    xBusy := FALSE;
                    step := 90;
                END_IF;
            END_IF;
        END_IF;

    80:
        xRetryTiming := TRUE;
        IF fbReconnect.Q THEN
            xRetryTiming := FALSE;
            step := 10;
        END_IF;

    90:
        IF xError THEN
            fbCore.CloseSocket();
        END_IF;

        IF xError AND (uiRetryCount < uiRetryMax) THEN
            uiRetryCount := uiRetryCount + 1;
            xError := FALSE;
            step := 80;
        ELSE
            xBusy := FALSE;
            step := 0;
        END_IF;
END_CASE;

(* ---- FB_SlmpReadDWordDevice.st ---- *)
FUNCTION_BLOCK FB_SlmpReadDWordDevice
VAR_INPUT
    xExecute         : BOOL;
    sIp              : STRING;
    uiPort           : UINT;
    udiHeadDevNo     : UDINT := 0;
    uiDeviceCode     : UINT := 16#00C2; // LTN
    uiPoints         : UINT := 1; // number of 2-word points
    tTimeout         : TIME := T#2S;
    uiRetryMax       : UINT := 2;
    tReconnectDelay  : TIME := T#500MS;
    xUse4E           : BOOL := FALSE;
    xUseUdp          : BOOL := FALSE;
    uiSerialNo       : UINT := 0;
END_VAR
VAR_OUTPUT
    xBusy            : BOOL;
    xDone            : BOOL;
    xError           : BOOL;
    diError          : DINT;
    uiRetryCount     : UINT;
    uiReadPoints     : UINT; // number of 2-word points
    udiValue0        : UDINT;
    aReadDWords      : ARRAY[0..SLMP_MAX_WORD_INDEX] OF UDINT;
    aLastResponse    : ARRAY[0..SLMP_LAST_RESPONSE_INDEX_MAX] OF BYTE;
    uiLastResponseLen: UINT;
    uiLastEndCode    : UINT;
END_VAR
VAR
    fbReadWord       : FB_SlmpReadWordDevice;
    uiPointsEff      : UINT := 0;
    idx              : UINT := 0;
    udiLow           : UDINT := 0;
    udiHigh          : UDINT := 0;
END_VAR

// === IMPLEMENTATION ===
uiPointsEff := uiPoints;
IF uiPointsEff > (SLMP_MAX_WORD_POINTS / 2) THEN
    uiPointsEff := SLMP_MAX_WORD_POINTS / 2;
END_IF;

fbReadWord(
    xExecute := xExecute,
    sIp := sIp,
    uiPort := uiPort,
    udiHeadDevNo := udiHeadDevNo,
    uiDeviceCode := uiDeviceCode,
    xAutoSubCommand := FALSE,
    uiSubCommand := SLMP_SUB_WORD2,
    uiPoints := uiPointsEff,
    tTimeout := tTimeout,
    uiRetryMax := uiRetryMax,
    tReconnectDelay := tReconnectDelay,
    xUse4E := xUse4E,
    xUseUdp := xUseUdp,
    uiSerialNo := uiSerialNo
);

xBusy := fbReadWord.xBusy;
xDone := fbReadWord.xDone;
xError := fbReadWord.xError;
diError := fbReadWord.diError;
uiRetryCount := fbReadWord.uiRetryCount;
uiLastResponseLen := fbReadWord.uiLastResponseLen;
uiLastEndCode := fbReadWord.uiLastEndCode;
FOR idx := 0 TO SLMP_LAST_RESPONSE_INDEX_MAX DO
    aLastResponse[idx] := fbReadWord.aLastResponse[idx];
END_FOR;

IF fbReadWord.xDone THEN
    uiReadPoints := uiPointsEff;
    FOR idx := 0 TO (uiPointsEff - 1) DO
        udiLow := TO_UDINT(fbReadWord.aValues[idx * 2]);
        udiHigh := TO_UDINT(fbReadWord.aValues[idx * 2 + 1]);
        aReadDWords[idx] := udiLow OR SHL(udiHigh, 16);
    END_FOR;
    IF uiPointsEff > 0 THEN
        udiValue0 := aReadDWords[0];
    END_IF;
END_IF;

(* ---- FB_SlmpReadPlcInfo.st ---- *)
FUNCTION_BLOCK FB_SlmpReadPlcInfo
VAR_INPUT
    xExecute         : BOOL;
    sIp              : STRING;
    uiPort           : UINT;
    tTimeout         : TIME := T#2S;
    uiRetryMax       : UINT := 2;
    tReconnectDelay  : TIME := T#500MS;
    xUse4E           : BOOL := FALSE;
    xUseUdp          : BOOL := FALSE;
    uiSerialNo       : UINT := 1;
END_VAR
VAR_OUTPUT
    xBusy            : BOOL;
    xDone            : BOOL;
    xError           : BOOL;
    diError          : DINT;
    uiRetryCount     : UINT;
    aCpuTypeNameRaw  : ARRAY[0..15] OF BYTE;
    uiCpuTypeCode    : UINT;
    xPlcRun          : BOOL;
    xPlcStop         : BOOL;
    uiPlcMode        : UINT; // 0: unknown, 1: run, 2: stop
    aLastResponse    : ARRAY[0..SLMP_LAST_RESPONSE_INDEX_MAX] OF BYTE;
    uiLastResponseLen: UINT;
    uiLastEndCode    : UINT;
    aLastResponseCpuInfo : ARRAY[0..SLMP_LAST_RESPONSE_INDEX_MAX] OF BYTE;
    uiLastResponseCpuInfoLen : UINT;
    uiLastEndCodeCpuInfo : UINT;
    aLastResponseSm403 : ARRAY[0..SLMP_LAST_RESPONSE_INDEX_MAX] OF BYTE;
    uiLastResponseSm403Len : UINT;
    uiLastEndCodeSm403 : UINT;
END_VAR
VAR
    step             : INT := 0;
    xExecPrev        : BOOL := FALSE;

    fbCore           : FB_SlmpCore;

    tx               : ARRAY[0..31] OF BYTE;
    rx               : ARRAY[0..SLMP_LAST_RESPONSE_INDEX_MAX] OF BYTE;
    txLen            : LINT := 0;
    rxLen            : LINT := 0;
    lenReq           : UINT := 0;
    endCode          : UINT := 0;
    byModeData       : BYTE := 0;

    iDataStart       : DINT := 11;
    iEndCodeStart    : DINT := 9;
    iNeedRxLen       : LINT := 0;
    idx              : UINT := 0;
    uiCopyLen        : UINT := 0;

    xStateTimeout    : BOOL := FALSE;
    xRetryTiming     : BOOL := FALSE;
    fbTimeout        : TON;
    fbReconnect      : TON;
END_VAR

// === IMPLEMENTATION ===
IF (xExecute AND NOT xExecPrev) THEN
    xBusy := TRUE;
    xDone := FALSE;
    xError := FALSE;
    diError := 0;
    uiRetryCount := 0;
    uiCpuTypeCode := 0;
    xPlcRun := FALSE;
    xPlcStop := FALSE;
    uiPlcMode := 0;
    uiLastResponseLen := 0;
    uiLastEndCode := 0;
    uiLastResponseCpuInfoLen := 0;
    uiLastEndCodeCpuInfo := 0;
    uiLastResponseSm403Len := 0;
    uiLastEndCodeSm403 := 0;
    FOR idx := 0 TO 15 DO
        aCpuTypeNameRaw[idx] := 0;
    END_FOR;
    FOR idx := 0 TO SLMP_LAST_RESPONSE_INDEX_MAX DO
        aLastResponse[idx] := 0;
        aLastResponseCpuInfo[idx] := 0;
        aLastResponseSm403[idx] := 0;
    END_FOR;
    step := 10;
END_IF;
xExecPrev := xExecute;

xStateTimeout := (step = 20) OR (step = 40) OR (step = 50) OR (step = 60) OR (step = 70);
fbTimeout(IN := xStateTimeout, PT := tTimeout);
fbReconnect(IN := xRetryTiming, PT := tReconnectDelay);

IF (step <> 0) AND (step <> 80) AND fbTimeout.Q THEN
    diError := -3010;
    xError := TRUE;
    step := 90;
END_IF;

CASE step OF
    0:
        xRetryTiming := FALSE;

    10:
        step := 20;

    20:
        IF fbCore.OpenAndConnect(sIp := sIp, uiPort := uiPort, xUseUdp := xUseUdp) THEN
            step := 30;
        ELSE
            CASE fbCore.diLastError OF
                -1: diError := -3001;
                -2: diError := -3005;
                -3: diError := -3002;
            ELSE
                diError := -3002;
            END_CASE;
            xError := TRUE;
            step := 90;
        END_IF;

    30:
        lenReq := 6; // monitor timer(2) + command(2) + subcommand(2)

        IF xUse4E THEN
            iDataStart := 15;
            iEndCodeStart := 13;
            tx[0] := 16#54; tx[1] := 16#00;
            tx[2] := TO_BYTE(uiSerialNo AND 16#00FF);
            tx[3] := TO_BYTE(SHR(uiSerialNo, 8) AND 16#00FF);
            tx[4] := 16#00; tx[5] := 16#00;
            tx[6] := 16#00;
            tx[7] := 16#FF;
            tx[8] := 16#FF; tx[9] := 16#03;
            tx[10] := 16#00;
            tx[11] := TO_BYTE(lenReq AND 16#00FF);
            tx[12] := TO_BYTE(SHR(lenReq, 8) AND 16#00FF);
            tx[13] := 16#10; tx[14] := 16#00;
            tx[15] := 16#01; tx[16] := 16#01;
            tx[17] := 16#00; tx[18] := 16#00;
            txLen := 19;
        ELSE
            iDataStart := 11;
            iEndCodeStart := 9;
            tx[0] := 16#50; tx[1] := 16#00;
            tx[2] := 16#00;
            tx[3] := 16#FF;
            tx[4] := 16#FF; tx[5] := 16#03;
            tx[6] := 16#00;
            tx[7] := TO_BYTE(lenReq AND 16#00FF);
            tx[8] := TO_BYTE(SHR(lenReq, 8) AND 16#00FF);
            tx[9] := 16#10; tx[10] := 16#00;
            tx[11] := 16#01; tx[12] := 16#01;
            tx[13] := 16#00; tx[14] := 16#00;
            txLen := 15;
        END_IF;

        step := 40;

    40:
        IF NOT fbCore.SendBytes(pData := ADR(tx[0]), liLen := txLen) THEN
            diError := -3003;
            xError := TRUE;
            step := 90;
        ELSE
            step := 50;
        END_IF;

    50:
        rxLen := fbCore.RecvBytes(pData := ADR(rx[0]), liMaxLen := SIZEOF(rx));
        IF rxLen > 0 THEN
            // Auto-detect response frame type from subheader.
            IF (rxLen >= 15) AND (rx[0] = 16#D4) AND (rx[1] = 16#00) THEN
                iDataStart := 15;
                iEndCodeStart := 13;
            ELSIF (rxLen >= 11) AND (rx[0] = 16#D0) AND (rx[1] = 16#00) THEN
                iDataStart := 11;
                iEndCodeStart := 9;
            END_IF;
            uiCopyLen := 0;
            IF rxLen > TO_LINT(SLMP_LAST_RESPONSE_INDEX_MAX + 1) THEN
                uiCopyLen := SLMP_LAST_RESPONSE_INDEX_MAX + 1;
            ELSE
                uiCopyLen := TO_UINT(rxLen);
            END_IF;
            uiLastResponseLen := uiCopyLen;
            uiLastResponseCpuInfoLen := uiCopyLen;
            IF uiCopyLen > 0 THEN
                FOR idx := 0 TO (uiCopyLen - 1) DO
                    aLastResponse[idx] := rx[idx];
                    aLastResponseCpuInfo[idx] := rx[idx];
                END_FOR;
            END_IF;
            iNeedRxLen := TO_LINT(iEndCodeStart) + 2;
            IF rxLen < iNeedRxLen THEN
                diError := -3004;
                xError := TRUE;
                step := 90;
            ELSE
                IF iEndCodeStart = 13 THEN
                    IF (TO_UINT(rx[2]) OR SHL(TO_UINT(rx[3]), 8)) <> uiSerialNo THEN
                        // Drop stale frame and keep waiting until timeout.
                        rxLen := 0;
                        uiLastResponseLen := 0;
                        uiLastResponseCpuInfoLen := 0;
                    END_IF;
                END_IF;
            END_IF;
            IF (NOT xError) AND (rxLen > 0) THEN
                endCode := TO_UINT(rx[iEndCodeStart]) OR SHL(TO_UINT(rx[iEndCodeStart + 1]), 8);
                uiLastEndCode := endCode;
                uiLastEndCodeCpuInfo := endCode;
                IF endCode <> 0 THEN
                    diError := TO_DINT(endCode);
                    xError := TRUE;
                    step := 90;
                ELSE
                    iNeedRxLen := TO_LINT(iDataStart) + 18; // 16-byte name + 2-byte code
                    IF rxLen < iNeedRxLen THEN
                        diError := -3004;
                        xError := TRUE;
                        step := 90;
                    ELSE
                        FOR idx := 0 TO 15 DO
                            aCpuTypeNameRaw[idx] := rx[iDataStart + TO_DINT(idx)];
                        END_FOR;
                        uiCpuTypeCode := TO_UINT(rx[iDataStart + 16]) OR SHL(TO_UINT(rx[iDataStart + 17]), 8);
                        step := 60;
                    END_IF;
                END_IF;
            END_IF;
        END_IF;

    60:
        lenReq := 12;
        IF xUse4E THEN
            iDataStart := 15;
            iEndCodeStart := 13;
            tx[0] := 16#54; tx[1] := 16#00;
            tx[2] := TO_BYTE(uiSerialNo AND 16#00FF);
            tx[3] := TO_BYTE(SHR(uiSerialNo, 8) AND 16#00FF);
            tx[4] := 16#00; tx[5] := 16#00;
            tx[6] := 16#00;
            tx[7] := 16#FF;
            tx[8] := 16#FF; tx[9] := 16#03;
            tx[10] := 16#00;
            tx[11] := TO_BYTE(lenReq AND 16#00FF);
            tx[12] := TO_BYTE(SHR(lenReq, 8) AND 16#00FF);
            tx[13] := 16#10; tx[14] := 16#00;
            tx[15] := 16#01; tx[16] := 16#04;
            tx[17] := 16#01; tx[18] := 16#00;
            tx[19] := TO_BYTE(403 AND 16#000000FF);
            tx[20] := TO_BYTE(SHR(403, 8) AND 16#000000FF);
            tx[21] := TO_BYTE(SHR(403, 16) AND 16#000000FF);
            tx[22] := TO_BYTE(SLMP_DEV_SM AND 16#00FF);
            tx[23] := 16#01;
            tx[24] := 16#00;
            txLen := 25;
        ELSE
            iDataStart := 11;
            iEndCodeStart := 9;
            tx[0] := 16#50; tx[1] := 16#00;
            tx[2] := 16#00;
            tx[3] := 16#FF;
            tx[4] := 16#FF; tx[5] := 16#03;
            tx[6] := 16#00;
            tx[7] := TO_BYTE(lenReq AND 16#00FF);
            tx[8] := TO_BYTE(SHR(lenReq, 8) AND 16#00FF);
            tx[9] := 16#10; tx[10] := 16#00;
            tx[11] := 16#01; tx[12] := 16#04;
            tx[13] := 16#01; tx[14] := 16#00;
            tx[15] := TO_BYTE(403 AND 16#000000FF);
            tx[16] := TO_BYTE(SHR(403, 8) AND 16#000000FF);
            tx[17] := TO_BYTE(SHR(403, 16) AND 16#000000FF);
            tx[18] := TO_BYTE(SLMP_DEV_SM AND 16#00FF);
            tx[19] := 16#01;
            tx[20] := 16#00;
            txLen := 21;
        END_IF;

        IF NOT fbCore.SendBytes(pData := ADR(tx[0]), liLen := txLen) THEN
            diError := -3003;
            xError := TRUE;
            step := 90;
        ELSE
            step := 70;
        END_IF;

    70:
        rxLen := fbCore.RecvBytes(pData := ADR(rx[0]), liMaxLen := SIZEOF(rx));
        IF rxLen > 0 THEN
            // Auto-detect response frame type from subheader.
            IF (rxLen >= 15) AND (rx[0] = 16#D4) AND (rx[1] = 16#00) THEN
                iDataStart := 15;
                iEndCodeStart := 13;
            ELSIF (rxLen >= 11) AND (rx[0] = 16#D0) AND (rx[1] = 16#00) THEN
                iDataStart := 11;
                iEndCodeStart := 9;
            END_IF;
            uiCopyLen := 0;
            IF rxLen > TO_LINT(SLMP_LAST_RESPONSE_INDEX_MAX + 1) THEN
                uiCopyLen := SLMP_LAST_RESPONSE_INDEX_MAX + 1;
            ELSE
                uiCopyLen := TO_UINT(rxLen);
            END_IF;
            uiLastResponseLen := uiCopyLen;
            uiLastResponseSm403Len := uiCopyLen;
            IF uiCopyLen > 0 THEN
                FOR idx := 0 TO (uiCopyLen - 1) DO
                    aLastResponse[idx] := rx[idx];
                    aLastResponseSm403[idx] := rx[idx];
                END_FOR;
            END_IF;
            iNeedRxLen := TO_LINT(iEndCodeStart) + 2;
            IF rxLen < iNeedRxLen THEN
                diError := -3004;
                xError := TRUE;
                step := 90;
            ELSE
                IF iEndCodeStart = 13 THEN
                    IF (TO_UINT(rx[2]) OR SHL(TO_UINT(rx[3]), 8)) <> uiSerialNo THEN
                        // Drop stale frame and keep waiting until timeout.
                        rxLen := 0;
                        uiLastResponseLen := 0;
                        uiLastResponseSm403Len := 0;
                    END_IF;
                END_IF;
            END_IF;
            IF (NOT xError) AND (rxLen > 0) THEN
                endCode := TO_UINT(rx[iEndCodeStart]) OR SHL(TO_UINT(rx[iEndCodeStart + 1]), 8);
                uiLastEndCode := endCode;
                uiLastEndCodeSm403 := endCode;
                IF endCode <> 0 THEN
                    diError := TO_DINT(endCode);
                    xError := TRUE;
                    step := 90;
                ELSE
                    iNeedRxLen := TO_LINT(iDataStart) + 1;
                    IF rxLen < iNeedRxLen THEN
                        diError := -3004;
                        xError := TRUE;
                        step := 90;
                    ELSE
                        byModeData := rx[iDataStart];
                        xPlcRun := (byModeData AND 16#F0) <> 0;
                        xPlcStop := NOT xPlcRun;
                        IF xPlcRun THEN
                            uiPlcMode := 1;
                        ELSE
                            uiPlcMode := 2;
                        END_IF;
                        xDone := TRUE;
                        xBusy := FALSE;
                        step := 90;
                    END_IF;
                END_IF;
            END_IF;
        END_IF;

    80:
        xRetryTiming := TRUE;
        IF fbReconnect.Q THEN
            xRetryTiming := FALSE;
            step := 10;
        END_IF;

    90:
        IF xError THEN
            fbCore.CloseSocket();
        END_IF;

        IF xError AND (uiRetryCount < uiRetryMax) THEN
            uiRetryCount := uiRetryCount + 1;
            xError := FALSE;
            step := 80;
        ELSE
            xBusy := FALSE;
            step := 0;
        END_IF;
END_CASE;

(* ---- FB_SlmpReadPlcInfoService.st ---- *)
FUNCTION_BLOCK FB_SlmpReadPlcInfoService
VAR_INPUT
    xExecute        : BOOL;
    sIp             : STRING;
    uiPort          : UINT;
    tTimeout        : TIME := T#2S;
    uiRetryMax      : UINT := 2;
    tReconnectDelay : TIME := T#500MS;
    xUse4E          : BOOL := FALSE;
    xUseUdp         : BOOL := FALSE;
    uiSerialNo      : UINT := 1;
END_VAR
VAR_OUTPUT
    xBusy           : BOOL;
    xDone           : BOOL;
    xError          : BOOL;
    diError         : DINT;
    uiRetryCount    : UINT;
    aPlcTypeNameRaw : ARRAY[0..15] OF BYTE;
    sPlcTypeName    : STRING(16);
    uiPlcTypeCode   : UINT;
    xPlcRun         : BOOL;
    xPlcStop        : BOOL;
    uiPlcMode       : UINT;
    aLastResponse   : ARRAY[0..SLMP_LAST_RESPONSE_INDEX_MAX] OF BYTE;
    uiLastResponseLen : UINT;
    uiLastEndCode   : UINT;
END_VAR
VAR
    fbReadPlcInfo   : FB_SlmpReadPlcInfo;
    udInstanceId    : UDINT := 0;

    xExecPrev       : BOOL := FALSE;
    xPending        : BOOL := FALSE;
    xActive         : BOOL := FALSE;
    xExecPulse      : BOOL := FALSE;
    iLockIdx        : INT := -1;
    uiSerialActive  : UINT := 0;

    idx             : UINT;
    uiSerialEff     : UINT;
    iSlot           : INT;
    iFreeSlot       : INT;
    xLocked         : BOOL;
    pTypeName       : POINTER TO BYTE;
    uiNameLen       : UINT;
END_VAR

// === IMPLEMENTATION ===
IF udInstanceId = 0 THEN
    GVL_SlmpRuntime.g_udServiceInstanceCounter := GVL_SlmpRuntime.g_udServiceInstanceCounter + 1;
    udInstanceId := GVL_SlmpRuntime.g_udServiceInstanceCounter;
    IF udInstanceId = 0 THEN
        udInstanceId := 1;
    END_IF;
END_IF;

IF xExecute AND (NOT xExecPrev) THEN
    IF (NOT xPending) AND (NOT xActive) THEN
        xDone := FALSE;
        xError := FALSE;
        diError := 0;
        uiRetryCount := 0;
        xPending := TRUE;
    END_IF;
END_IF;
xExecPrev := xExecute;

xExecPulse := FALSE;
IF xPending AND (NOT xActive) THEN
    xLocked := FALSE;
    iFreeSlot := -1;
    FOR iSlot := 0 TO 7 DO
        IF (GVL_SlmpRuntime.g_aLockOwner[iSlot] <> 0) AND
           (GVL_SlmpRuntime.g_aLockIp[iSlot] = sIp) AND
           (GVL_SlmpRuntime.g_aLockPort[iSlot] = uiPort) AND
           (GVL_SlmpRuntime.g_aLockUseUdp[iSlot] = xUseUdp) THEN
            xLocked := TRUE;
            EXIT;
        END_IF;
        IF (iFreeSlot < 0) AND (GVL_SlmpRuntime.g_aLockOwner[iSlot] = 0) THEN
            iFreeSlot := iSlot;
        END_IF;
    END_FOR;

    IF (NOT xLocked) AND (iFreeSlot >= 0) THEN
        GVL_SlmpRuntime.g_aLockOwner[iFreeSlot] := udInstanceId;
        GVL_SlmpRuntime.g_aLockIp[iFreeSlot] := sIp;
        GVL_SlmpRuntime.g_aLockPort[iFreeSlot] := uiPort;
        GVL_SlmpRuntime.g_aLockUseUdp[iFreeSlot] := xUseUdp;
        iLockIdx := iFreeSlot;

        xActive := TRUE;
        xExecPulse := TRUE;
        IF xUse4E THEN
            uiSerialActive := F_SlmpNextSerialNo(uiSeed := uiSerialNo);
        END_IF;
    END_IF;
END_IF;

IF xActive THEN
    IF xUse4E THEN
        uiSerialEff := uiSerialActive;
        IF uiSerialEff = 0 THEN
            uiSerialEff := 1;
        END_IF;
    ELSE
        uiSerialEff := uiSerialNo;
    END_IF;

    fbReadPlcInfo(
        xExecute := xExecPulse,
        sIp := sIp,
        uiPort := uiPort,
        tTimeout := tTimeout,
        uiRetryMax := uiRetryMax,
        tReconnectDelay := tReconnectDelay,
        xUse4E := xUse4E,
        xUseUdp := xUseUdp,
        uiSerialNo := uiSerialEff
    );
ELSE
    xBusy := xPending;
    IF NOT xExecute THEN
        xDone := FALSE;
        xError := FALSE;
        diError := 0;
        uiRetryCount := 0;
    END_IF;
    RETURN;
END_IF;

xBusy := fbReadPlcInfo.xBusy;
xDone := fbReadPlcInfo.xDone;
xError := fbReadPlcInfo.xError;
diError := fbReadPlcInfo.diError;
uiRetryCount := fbReadPlcInfo.uiRetryCount;

IF fbReadPlcInfo.xDone THEN
    FOR idx := 0 TO 15 DO
        aPlcTypeNameRaw[idx] := fbReadPlcInfo.aCpuTypeNameRaw[idx];
    END_FOR;

    pTypeName := ADR(sPlcTypeName);
    FOR idx := 0 TO 16 DO
        pTypeName[idx] := 0;
    END_FOR;
    uiNameLen := 0;
    FOR idx := 0 TO 15 DO
        IF aPlcTypeNameRaw[idx] = 0 THEN
            EXIT;
        END_IF;
        pTypeName[uiNameLen] := aPlcTypeNameRaw[idx];
        uiNameLen := uiNameLen + 1;
    END_FOR;
    pTypeName[uiNameLen] := 0;

    uiPlcTypeCode := fbReadPlcInfo.uiCpuTypeCode;
    xPlcRun := fbReadPlcInfo.xPlcRun;
    xPlcStop := fbReadPlcInfo.xPlcStop;
    uiPlcMode := fbReadPlcInfo.uiPlcMode;

    FOR idx := 0 TO SLMP_LAST_RESPONSE_INDEX_MAX DO
        aLastResponse[idx] := fbReadPlcInfo.aLastResponse[idx];
    END_FOR;
    uiLastResponseLen := fbReadPlcInfo.uiLastResponseLen;
    uiLastEndCode := fbReadPlcInfo.uiLastEndCode;
END_IF;

IF fbReadPlcInfo.xDone OR fbReadPlcInfo.xError THEN
    xPending := FALSE;
    xActive := FALSE;
    IF iLockIdx >= 0 THEN
        GVL_SlmpRuntime.g_aLockOwner[iLockIdx] := 0;
        GVL_SlmpRuntime.g_aLockIp[iLockIdx] := '';
        GVL_SlmpRuntime.g_aLockPort[iLockIdx] := 0;
        GVL_SlmpRuntime.g_aLockUseUdp[iLockIdx] := FALSE;
        iLockIdx := -1;
    END_IF;
END_IF;

(* ---- FB_SlmpReadWordDevice.st ---- *)
FUNCTION_BLOCK FB_SlmpReadWordDevice
VAR_INPUT
    xExecute         : BOOL;
    sIp              : STRING;
    uiPort           : UINT;
    udiHeadDevNo     : UDINT := 100;
    uiDeviceCode     : UINT := 16#00A8; // D
    xAutoSubCommand  : BOOL := TRUE;
    uiSubCommand     : UINT := 16#0000;
    uiPoints         : UINT := 1;
    tTimeout         : TIME := T#2S;
    uiRetryMax       : UINT := 2;
    tReconnectDelay  : TIME := T#500MS;
    xUse4E           : BOOL := FALSE;
    xUseUdp          : BOOL := FALSE;
    uiSerialNo       : UINT := 0;
END_VAR
VAR_OUTPUT
    xBusy            : BOOL;
    xDone            : BOOL;
    xError           : BOOL;
    diError          : DINT;
    uiRetryCount     : UINT;
    uiReadWords      : UINT;
    uiValue0         : UINT;
    aValues          : ARRAY[0..SLMP_MAX_WORD_INDEX] OF UINT;
    aLastResponse    : ARRAY[0..SLMP_LAST_RESPONSE_INDEX_MAX] OF BYTE;
    uiLastResponseLen: UINT;
    uiLastEndCode    : UINT;
END_VAR
VAR
    step             : INT := 0;
    xExecPrev        : BOOL := FALSE;

    fbCore           : FB_SlmpCore;

    tx               : ARRAY[0..31] OF BYTE;
    rx               : ARRAY[0..SLMP_READ_RX_INDEX_MAX] OF BYTE;
    txLen            : LINT := 0;
    rxLen            : LINT := 0;
    lenReq           : UINT := 0;
    endCode          : UINT := 0;

    uiPointsReq      : UINT := 0;
    uiPointsEff      : UINT := 0;
    uiPointsProto    : UINT := 0;
    uiSubCmdEff      : UINT := 0;
    xWord2Mode       : BOOL := FALSE;
    iDataStart       : DINT := 11;
    iEndCodeStart    : DINT := 9;
    iNeedRxLen       : LINT := 0;
    uiRxSerialNo     : UINT := 0;
    uiCopyLen        : UINT := 0;
    idx              : UINT := 0;

    xStateTimeout    : BOOL := FALSE;
    xRetryTiming     : BOOL := FALSE;
    fbTimeout        : TON;
    fbReconnect      : TON;
END_VAR

// === IMPLEMENTATION ===
IF (xExecute AND NOT xExecPrev) THEN
    xBusy := TRUE;
    xDone := FALSE;
    xError := FALSE;
    diError := 0;
    uiRetryCount := 0;
    uiReadWords := 0;
    uiValue0 := 0;
    uiLastResponseLen := 0;
    uiLastEndCode := 0;
    FOR idx := 0 TO SLMP_MAX_WORD_INDEX DO
        aValues[idx] := 0;
    END_FOR;
    FOR idx := 0 TO SLMP_LAST_RESPONSE_INDEX_MAX DO
        aLastResponse[idx] := 0;
    END_FOR;
    step := 10;
END_IF;
xExecPrev := xExecute;

xStateTimeout := (step = 20) OR (step = 40) OR (step = 50);
fbTimeout(IN := xStateTimeout, PT := tTimeout);
fbReconnect(IN := xRetryTiming, PT := tReconnectDelay);

IF (step <> 0) AND (step <> 80) AND fbTimeout.Q THEN
    diError := -1010;
    xError := TRUE;
    step := 90;
END_IF;

CASE step OF
    0:
        xRetryTiming := FALSE;

    10:
        uiSubCmdEff := F_SlmpResolveSubCommand(
            uiDeviceCode := uiDeviceCode,
            xAutoSubCommand := xAutoSubCommand,
            uiSubCommand := uiSubCommand
        );
        xWord2Mode := (uiSubCmdEff = SLMP_SUB_WORD2);

        uiPointsReq := uiPoints;
        IF uiPointsReq = 0 THEN
            diError := -1000;
            xError := TRUE;
            xBusy := FALSE;
            step := 0;
        ELSE
            uiPointsEff := F_SlmpClampPoints(uiPoints := uiPointsReq, xBitMode := FALSE);
            IF xWord2Mode THEN
                IF uiPointsEff > (SLMP_MAX_WORD_POINTS / 2) THEN
                    uiPointsEff := SLMP_MAX_WORD_POINTS / 2;
                END_IF;
                uiPointsProto := uiPointsEff * 2;
            ELSE
                uiPointsProto := uiPointsEff;
            END_IF;
        END_IF;

        IF NOT xError THEN
            step := 20;
        END_IF;

    20:
        IF fbCore.OpenAndConnect(sIp := sIp, uiPort := uiPort, xUseUdp := xUseUdp) THEN
            step := 30;
        ELSE
            CASE fbCore.diLastError OF
                -1: diError := -1001;
                -2: diError := -1005;
                -3: diError := -1002;
            ELSE
                diError := -1002;
            END_CASE;
            xError := TRUE;
            step := 90;
        END_IF;

    30:
        lenReq := 12;
        IF xUse4E THEN
            iDataStart := 15;
            iEndCodeStart := 13;
            tx[0] := 16#54; tx[1] := 16#00;
            tx[2] := TO_BYTE(uiSerialNo AND 16#00FF);
            tx[3] := TO_BYTE(SHR(uiSerialNo, 8) AND 16#00FF);
            tx[4] := 16#00; tx[5] := 16#00;
            tx[6] := 16#00;
            tx[7] := 16#FF;
            tx[8] := 16#FF; tx[9] := 16#03;
            tx[10] := 16#00;
            tx[11] := TO_BYTE(lenReq AND 16#00FF);
            tx[12] := TO_BYTE(SHR(lenReq, 8) AND 16#00FF);
            tx[13] := 16#10; tx[14] := 16#00;
            tx[15] := 16#01; tx[16] := 16#04;
            tx[17] := TO_BYTE(uiSubCmdEff AND 16#00FF);
            tx[18] := TO_BYTE(SHR(uiSubCmdEff, 8) AND 16#00FF);
            tx[19] := TO_BYTE(udiHeadDevNo AND 16#000000FF);
            tx[20] := TO_BYTE(SHR(udiHeadDevNo, 8) AND 16#000000FF);
            tx[21] := TO_BYTE(SHR(udiHeadDevNo, 16) AND 16#000000FF);
            tx[22] := TO_BYTE(uiDeviceCode AND 16#00FF);
            tx[23] := TO_BYTE(uiPointsProto AND 16#00FF);
            tx[24] := TO_BYTE(SHR(uiPointsProto, 8) AND 16#00FF);
            txLen := 25;
        ELSE
            iDataStart := 11;
            iEndCodeStart := 9;
            tx[0] := 16#50; tx[1] := 16#00;
            tx[2] := 16#00;
            tx[3] := 16#FF;
            tx[4] := 16#FF; tx[5] := 16#03;
            tx[6] := 16#00;
            tx[7] := TO_BYTE(lenReq AND 16#00FF);
            tx[8] := TO_BYTE(SHR(lenReq, 8) AND 16#00FF);
            tx[9] := 16#10; tx[10] := 16#00;
            tx[11] := 16#01; tx[12] := 16#04;
            tx[13] := TO_BYTE(uiSubCmdEff AND 16#00FF);
            tx[14] := TO_BYTE(SHR(uiSubCmdEff, 8) AND 16#00FF);
            tx[15] := TO_BYTE(udiHeadDevNo AND 16#000000FF);
            tx[16] := TO_BYTE(SHR(udiHeadDevNo, 8) AND 16#000000FF);
            tx[17] := TO_BYTE(SHR(udiHeadDevNo, 16) AND 16#000000FF);
            tx[18] := TO_BYTE(uiDeviceCode AND 16#00FF);
            tx[19] := TO_BYTE(uiPointsProto AND 16#00FF);
            tx[20] := TO_BYTE(SHR(uiPointsProto, 8) AND 16#00FF);
            txLen := 21;
        END_IF;
        step := 40;

    40:
        IF NOT fbCore.SendBytes(pData := ADR(tx[0]), liLen := txLen) THEN
            diError := -1003;
            xError := TRUE;
            step := 90;
        ELSE
            step := 50;
        END_IF;

    50:
        rxLen := fbCore.RecvBytes(pData := ADR(rx[0]), liMaxLen := SIZEOF(rx));
        IF rxLen > 0 THEN
            uiCopyLen := 0;
            IF rxLen > TO_LINT(SLMP_LAST_RESPONSE_INDEX_MAX + 1) THEN
                uiCopyLen := SLMP_LAST_RESPONSE_INDEX_MAX + 1;
            ELSE
                uiCopyLen := TO_UINT(rxLen);
            END_IF;
            uiLastResponseLen := uiCopyLen;
            IF uiCopyLen > 0 THEN
                FOR idx := 0 TO (uiCopyLen - 1) DO
                    aLastResponse[idx] := rx[idx];
                END_FOR;
            END_IF;

            IF xWord2Mode THEN
                iNeedRxLen := iDataStart + TO_LINT(uiPointsEff) * 4;
            ELSE
                iNeedRxLen := iDataStart + TO_LINT(uiPointsEff) * 2;
            END_IF;
            IF rxLen < iNeedRxLen THEN
                diError := -1004;
                xError := TRUE;
                step := 90;
            ELSE
                IF xUse4E THEN
                    uiRxSerialNo := TO_UINT(rx[2]) OR SHL(TO_UINT(rx[3]), 8);
                    IF uiRxSerialNo <> uiSerialNo THEN
                        // Drop stale frame and keep waiting until timeout.
                        rxLen := 0;
                        uiLastResponseLen := 0;
                    END_IF;
                END_IF;
            END_IF;
            IF (NOT xError) AND (rxLen > 0) THEN
                endCode := TO_UINT(rx[iEndCodeStart]) OR SHL(TO_UINT(rx[iEndCodeStart + 1]), 8);
                uiLastEndCode := endCode;
                IF endCode <> 0 THEN
                    diError := TO_DINT(endCode);
                    xError := TRUE;
                    step := 90;
                ELSE
                    IF xWord2Mode THEN
                        FOR idx := 0 TO (uiPointsEff - 1) DO
                            aValues[idx * 2] := TO_UINT(rx[iDataStart + TO_DINT(idx) * 4]) OR
                                SHL(TO_UINT(rx[iDataStart + TO_DINT(idx) * 4 + 1]), 8);
                            aValues[idx * 2 + 1] := TO_UINT(rx[iDataStart + TO_DINT(idx) * 4 + 2]) OR
                                SHL(TO_UINT(rx[iDataStart + TO_DINT(idx) * 4 + 3]), 8);
                        END_FOR;
                        uiReadWords := uiPointsEff * 2;
                    ELSE
                        FOR idx := 0 TO (uiPointsEff - 1) DO
                            aValues[idx] := TO_UINT(rx[iDataStart + TO_DINT(idx) * 2]) OR
                                SHL(TO_UINT(rx[iDataStart + TO_DINT(idx) * 2 + 1]), 8);
                        END_FOR;
                        uiReadWords := uiPointsEff;
                    END_IF;
                    uiValue0 := aValues[0];
                    xDone := TRUE;
                    xBusy := FALSE;
                    step := 90;
                END_IF;
            END_IF;
        END_IF;

    80:
        xRetryTiming := TRUE;
        IF fbReconnect.Q THEN
            xRetryTiming := FALSE;
            step := 10;
        END_IF;

    90:
        IF xError THEN
            fbCore.CloseSocket();
        END_IF;

        IF xError AND (uiRetryCount < uiRetryMax) THEN
            uiRetryCount := uiRetryCount + 1;
            xError := FALSE;
            step := 80;
        ELSE
            xBusy := FALSE;
            step := 0;
        END_IF;
END_CASE;

(* ---- FB_SlmpReadWordService.st ---- *)
FUNCTION_BLOCK FB_SlmpReadWordService
VAR_INPUT
    xExecute        : BOOL;
    sIp             : STRING;
    uiPort          : UINT;
    udiHeadDevNo    : UDINT;
    uiDeviceCode    : UINT;
    uiPoints        : UINT;
    tTimeout        : TIME := T#2S;
    uiRetryMax      : UINT := 2;
    tReconnectDelay : TIME := T#500MS;
    xUse4E          : BOOL := FALSE;
    xUseUdp         : BOOL := FALSE;
    uiSerialNo      : UINT := 1;
END_VAR
VAR_OUTPUT
    xBusy           : BOOL;
    xDone           : BOOL;
    xError          : BOOL;
    diError         : DINT;
    uiRetryCount    : UINT;
    uiReadWords     : UINT;
    uiValue0        : UINT;
    aReadValues     : ARRAY[0..SLMP_MAX_WORD_INDEX] OF UINT;
    aLastResponse   : ARRAY[0..SLMP_LAST_RESPONSE_INDEX_MAX] OF BYTE;
    uiLastResponseLen : UINT;
    uiLastEndCode   : UINT;
END_VAR
VAR
    fbReadWord      : FB_SlmpReadWordDevice;
    udInstanceId    : UDINT := 0;

    xExecPrev       : BOOL := FALSE;
    xPending        : BOOL := FALSE;
    xActive         : BOOL := FALSE;
    xExecPulse      : BOOL := FALSE;
    iLockIdx        : INT := -1;

    udiHeadLatched  : UDINT := 0;
    uiDeviceLatched : UINT := 0;
    uiPointsLatched : UINT := 0;
    uiSerialActive  : UINT := 0;

    idx             : UINT;
    uiSerialEff     : UINT;
    iSlot           : INT;
    iFreeSlot       : INT;
    xLocked         : BOOL;
END_VAR

// === IMPLEMENTATION ===
IF udInstanceId = 0 THEN
    GVL_SlmpRuntime.g_udServiceInstanceCounter := GVL_SlmpRuntime.g_udServiceInstanceCounter + 1;
    udInstanceId := GVL_SlmpRuntime.g_udServiceInstanceCounter;
    IF udInstanceId = 0 THEN
        udInstanceId := 1;
    END_IF;
END_IF;

IF xExecute AND (NOT xExecPrev) THEN
    IF (NOT xPending) AND (NOT xActive) THEN
        udiHeadLatched := udiHeadDevNo;
        uiDeviceLatched := uiDeviceCode;
        uiPointsLatched := uiPoints;
        xDone := FALSE;
        xError := FALSE;
        diError := 0;
        uiRetryCount := 0;
        xPending := TRUE;
    END_IF;
END_IF;
xExecPrev := xExecute;

xExecPulse := FALSE;
IF xPending AND (NOT xActive) THEN
    xLocked := FALSE;
    iFreeSlot := -1;
    FOR iSlot := 0 TO 7 DO
        IF (GVL_SlmpRuntime.g_aLockOwner[iSlot] <> 0) AND
           (GVL_SlmpRuntime.g_aLockIp[iSlot] = sIp) AND
           (GVL_SlmpRuntime.g_aLockPort[iSlot] = uiPort) AND
           (GVL_SlmpRuntime.g_aLockUseUdp[iSlot] = xUseUdp) THEN
            xLocked := TRUE;
            EXIT;
        END_IF;
        IF (iFreeSlot < 0) AND (GVL_SlmpRuntime.g_aLockOwner[iSlot] = 0) THEN
            iFreeSlot := iSlot;
        END_IF;
    END_FOR;

    IF (NOT xLocked) AND (iFreeSlot >= 0) THEN
        GVL_SlmpRuntime.g_aLockOwner[iFreeSlot] := udInstanceId;
        GVL_SlmpRuntime.g_aLockIp[iFreeSlot] := sIp;
        GVL_SlmpRuntime.g_aLockPort[iFreeSlot] := uiPort;
        GVL_SlmpRuntime.g_aLockUseUdp[iFreeSlot] := xUseUdp;
        iLockIdx := iFreeSlot;

        xActive := TRUE;
        xExecPulse := TRUE;
        IF xUse4E THEN
            uiSerialActive := F_SlmpNextSerialNo(uiSeed := uiSerialNo);
        END_IF;
    END_IF;
END_IF;

IF xActive THEN
    IF xUse4E THEN
        uiSerialEff := uiSerialActive;
        IF uiSerialEff = 0 THEN
            uiSerialEff := 1;
        END_IF;
    ELSE
        uiSerialEff := uiSerialNo;
    END_IF;

    fbReadWord(
        xExecute := xExecPulse,
        sIp := sIp,
        uiPort := uiPort,
        udiHeadDevNo := udiHeadLatched,
        uiDeviceCode := uiDeviceLatched,
        xAutoSubCommand := TRUE,
        uiSubCommand := 0,
        uiPoints := uiPointsLatched,
        tTimeout := tTimeout,
        uiRetryMax := uiRetryMax,
        tReconnectDelay := tReconnectDelay,
        xUse4E := xUse4E,
        xUseUdp := xUseUdp,
        uiSerialNo := uiSerialEff
    );
ELSE
    xBusy := xPending;
    IF NOT xExecute THEN
        xDone := FALSE;
        xError := FALSE;
        diError := 0;
        uiRetryCount := 0;
    END_IF;
    RETURN;
END_IF;

xBusy := fbReadWord.xBusy;
xDone := fbReadWord.xDone;
xError := fbReadWord.xError;
diError := fbReadWord.diError;
uiRetryCount := fbReadWord.uiRetryCount;

IF fbReadWord.xDone THEN
    uiReadWords := fbReadWord.uiReadWords;
    uiValue0 := fbReadWord.uiValue0;
    FOR idx := 0 TO SLMP_MAX_WORD_INDEX DO
        aReadValues[idx] := fbReadWord.aValues[idx];
    END_FOR;
    FOR idx := 0 TO SLMP_LAST_RESPONSE_INDEX_MAX DO
        aLastResponse[idx] := fbReadWord.aLastResponse[idx];
    END_FOR;
    uiLastResponseLen := fbReadWord.uiLastResponseLen;
    uiLastEndCode := fbReadWord.uiLastEndCode;
END_IF;

IF fbReadWord.xDone OR fbReadWord.xError THEN
    xPending := FALSE;
    xActive := FALSE;
    IF iLockIdx >= 0 THEN
        GVL_SlmpRuntime.g_aLockOwner[iLockIdx] := 0;
        GVL_SlmpRuntime.g_aLockIp[iLockIdx] := '';
        GVL_SlmpRuntime.g_aLockPort[iLockIdx] := 0;
        GVL_SlmpRuntime.g_aLockUseUdp[iLockIdx] := FALSE;
        iLockIdx := -1;
    END_IF;
END_IF;

(* ---- FB_SlmpWriteBitDevice.st ---- *)
FUNCTION_BLOCK FB_SlmpWriteBitDevice
VAR_INPUT
    xExecute         : BOOL;
    sIp              : STRING;
    uiPort           : UINT;
    udiHeadDevNo     : UDINT := 100;
    uiDeviceCode     : UINT := 16#0090; // M
    xAutoSubCommand  : BOOL := TRUE;
    uiSubCommand     : UINT := 16#0001;
    uiPoints         : UINT := 1;
    aWriteBits       : ARRAY[0..SLMP_MAX_BIT_INDEX] OF BOOL;
    tTimeout         : TIME := T#2S;
    uiRetryMax       : UINT := 2;
    tReconnectDelay  : TIME := T#500MS;
    xUse4E           : BOOL := FALSE;
    xUseUdp          : BOOL := FALSE;
    uiSerialNo       : UINT := 0;
END_VAR
VAR_OUTPUT
    xBusy            : BOOL;
    xDone            : BOOL;
    xError           : BOOL;
    diError          : DINT;
    uiRetryCount     : UINT;
    aLastResponse    : ARRAY[0..SLMP_LAST_RESPONSE_INDEX_MAX] OF BYTE;
    uiLastResponseLen: UINT;
    uiLastEndCode    : UINT;
END_VAR
VAR
    step             : INT := 0;
    xExecPrev        : BOOL := FALSE;

    fbCore           : FB_SlmpCore;

    tx               : ARRAY[0..SLMP_WRITE_TX_INDEX_MAX] OF BYTE;
    rx               : ARRAY[0..SLMP_LAST_RESPONSE_INDEX_MAX] OF BYTE;
    txLen            : LINT := 0;
    rxLen            : LINT := 0;
    lenReq           : UINT := 0;
    endCode          : UINT := 0;

    uiPointsReq      : UINT := 0;
    uiPointsEff      : UINT := 0;
    uiSubCmdEff      : UINT := 0;
    idx              : UINT := 0;
    iDataStart       : DINT := 21;
    iEndCodeStart    : DINT := 9;
    iMinRxLen        : LINT := 11;
    uiRxSerialNo     : UINT := 0;
    uiCopyLen        : UINT := 0;
    iPayloadBytes    : LINT := 0;
    iByteOffset      : DINT := 0;

    xStateTimeout    : BOOL := FALSE;
    xRetryTiming     : BOOL := FALSE;
    fbTimeout        : TON;
    fbReconnect      : TON;
END_VAR

// === IMPLEMENTATION ===
IF (xExecute AND NOT xExecPrev) THEN
    xBusy := TRUE;
    xDone := FALSE;
    xError := FALSE;
    diError := 0;
    uiRetryCount := 0;
    uiLastResponseLen := 0;
    uiLastEndCode := 0;
    FOR idx := 0 TO SLMP_LAST_RESPONSE_INDEX_MAX DO
        aLastResponse[idx] := 0;
    END_FOR;
    step := 10;
END_IF;
xExecPrev := xExecute;

xStateTimeout := (step = 20) OR (step = 40) OR (step = 50);
fbTimeout(IN := xStateTimeout, PT := tTimeout);
fbReconnect(IN := xRetryTiming, PT := tReconnectDelay);

IF (step <> 0) AND (step <> 80) AND fbTimeout.Q THEN
    diError := -2010;
    xError := TRUE;
    step := 90;
END_IF;

CASE step OF
    0:
        xRetryTiming := FALSE;

    10:
        uiSubCmdEff := F_SlmpResolveSubCommand(
            uiDeviceCode := uiDeviceCode,
            xAutoSubCommand := xAutoSubCommand,
            uiSubCommand := uiSubCommand
        );

        uiPointsReq := uiPoints;
        IF uiPointsReq = 0 THEN
            diError := -2000;
            xError := TRUE;
            xBusy := FALSE;
            step := 0;
        ELSE
            uiPointsEff := F_SlmpClampPoints(uiPoints := uiPointsReq, xBitMode := TRUE);
        END_IF;

        IF NOT xError THEN
            step := 20;
        END_IF;

    20:
        IF fbCore.OpenAndConnect(sIp := sIp, uiPort := uiPort, xUseUdp := xUseUdp) THEN
            step := 30;
        ELSE
            CASE fbCore.diLastError OF
                -1: diError := -2001;
                -2: diError := -2005;
                -3: diError := -2002;
            ELSE
                diError := -2002;
            END_CASE;
            xError := TRUE;
            step := 90;
        END_IF;

    30:
        IF xUse4E THEN
            iDataStart := 25;
            iEndCodeStart := 13;
            iMinRxLen := 15;
        ELSE
            iDataStart := 21;
            iEndCodeStart := 9;
            iMinRxLen := 11;
        END_IF;

        iPayloadBytes := TO_LINT((uiPointsEff + 1) / 2);
        lenReq := TO_UINT(12 + TO_UINT(iPayloadBytes));

        IF xUse4E THEN
            tx[0] := 16#54; tx[1] := 16#00;
            tx[2] := TO_BYTE(uiSerialNo AND 16#00FF);
            tx[3] := TO_BYTE(SHR(uiSerialNo, 8) AND 16#00FF);
            tx[4] := 16#00; tx[5] := 16#00;
            tx[6] := 16#00;
            tx[7] := 16#FF;
            tx[8] := 16#FF; tx[9] := 16#03;
            tx[10] := 16#00;
            tx[11] := TO_BYTE(lenReq AND 16#00FF);
            tx[12] := TO_BYTE(SHR(lenReq, 8) AND 16#00FF);
            tx[13] := 16#10; tx[14] := 16#00;
            tx[15] := 16#01; tx[16] := 16#14;
            tx[17] := TO_BYTE(uiSubCmdEff AND 16#00FF);
            tx[18] := TO_BYTE(SHR(uiSubCmdEff, 8) AND 16#00FF);
            tx[19] := TO_BYTE(udiHeadDevNo AND 16#000000FF);
            tx[20] := TO_BYTE(SHR(udiHeadDevNo, 8) AND 16#000000FF);
            tx[21] := TO_BYTE(SHR(udiHeadDevNo, 16) AND 16#000000FF);
            tx[22] := TO_BYTE(uiDeviceCode AND 16#00FF);
            tx[23] := TO_BYTE(uiPointsEff AND 16#00FF);
            tx[24] := TO_BYTE(SHR(uiPointsEff, 8) AND 16#00FF);
        ELSE
            tx[0] := 16#50; tx[1] := 16#00;
            tx[2] := 16#00;
            tx[3] := 16#FF;
            tx[4] := 16#FF; tx[5] := 16#03;
            tx[6] := 16#00;
            tx[7] := TO_BYTE(lenReq AND 16#00FF);
            tx[8] := TO_BYTE(SHR(lenReq, 8) AND 16#00FF);
            tx[9] := 16#10; tx[10] := 16#00;
            tx[11] := 16#01; tx[12] := 16#14;
            tx[13] := TO_BYTE(uiSubCmdEff AND 16#00FF);
            tx[14] := TO_BYTE(SHR(uiSubCmdEff, 8) AND 16#00FF);
            tx[15] := TO_BYTE(udiHeadDevNo AND 16#000000FF);
            tx[16] := TO_BYTE(SHR(udiHeadDevNo, 8) AND 16#000000FF);
            tx[17] := TO_BYTE(SHR(udiHeadDevNo, 16) AND 16#000000FF);
            tx[18] := TO_BYTE(uiDeviceCode AND 16#00FF);
            tx[19] := TO_BYTE(uiPointsEff AND 16#00FF);
            tx[20] := TO_BYTE(SHR(uiPointsEff, 8) AND 16#00FF);
        END_IF;

        FOR idx := 0 TO ((uiPointsEff - 1) / 2) DO
            tx[iDataStart + TO_DINT(idx)] := 16#00;
        END_FOR;
        FOR idx := 0 TO (uiPointsEff - 1) DO
            iByteOffset := iDataStart + TO_DINT(idx / 2);
            IF aWriteBits[idx] THEN
                IF (idx MOD 2) = 0 THEN
                    tx[iByteOffset] := TO_BYTE(tx[iByteOffset] OR 16#10);
                ELSE
                    tx[iByteOffset] := TO_BYTE(tx[iByteOffset] OR 16#01);
                END_IF;
            END_IF;
        END_FOR;

        txLen := TO_LINT(iDataStart) + iPayloadBytes;
        step := 40;

    40:
        IF NOT fbCore.SendBytes(pData := ADR(tx[0]), liLen := txLen) THEN
            diError := -2003;
            xError := TRUE;
            step := 90;
        ELSE
            step := 50;
        END_IF;

    50:
        rxLen := fbCore.RecvBytes(pData := ADR(rx[0]), liMaxLen := SIZEOF(rx));
        IF rxLen > 0 THEN
            uiCopyLen := 0;
            IF rxLen > TO_LINT(SLMP_LAST_RESPONSE_INDEX_MAX + 1) THEN
                uiCopyLen := SLMP_LAST_RESPONSE_INDEX_MAX + 1;
            ELSE
                uiCopyLen := TO_UINT(rxLen);
            END_IF;
            uiLastResponseLen := uiCopyLen;
            IF uiCopyLen > 0 THEN
                FOR idx := 0 TO (uiCopyLen - 1) DO
                    aLastResponse[idx] := rx[idx];
                END_FOR;
            END_IF;
            IF rxLen < iMinRxLen THEN
                diError := -2004;
                xError := TRUE;
                step := 90;
            ELSE
                IF xUse4E THEN
                    uiRxSerialNo := TO_UINT(rx[2]) OR SHL(TO_UINT(rx[3]), 8);
                    IF uiRxSerialNo <> uiSerialNo THEN
                        // Drop stale frame and keep waiting until timeout.
                        rxLen := 0;
                        uiLastResponseLen := 0;
                    END_IF;
                END_IF;
            END_IF;
            IF (NOT xError) AND (rxLen > 0) THEN
                endCode := TO_UINT(rx[iEndCodeStart]) OR SHL(TO_UINT(rx[iEndCodeStart + 1]), 8);
                uiLastEndCode := endCode;
                IF endCode <> 0 THEN
                    diError := TO_DINT(endCode);
                    xError := TRUE;
                    step := 90;
                ELSE
                    xDone := TRUE;
                    xBusy := FALSE;
                    step := 90;
                END_IF;
            END_IF;
        END_IF;

    80:
        xRetryTiming := TRUE;
        IF fbReconnect.Q THEN
            xRetryTiming := FALSE;
            step := 10;
        END_IF;

    90:
        IF xError THEN
            fbCore.CloseSocket();
        END_IF;

        IF xError AND (uiRetryCount < uiRetryMax) THEN
            uiRetryCount := uiRetryCount + 1;
            xError := FALSE;
            step := 80;
        ELSE
            xBusy := FALSE;
            step := 0;
        END_IF;
END_CASE;

(* ---- FB_SlmpWriteBitService.st ---- *)
FUNCTION_BLOCK FB_SlmpWriteBitService
VAR_INPUT
    xExecute        : BOOL;
    sIp             : STRING;
    uiPort          : UINT;
    udiHeadDevNo    : UDINT;
    uiDeviceCode    : UINT;
    uiPoints        : UINT;
    tTimeout        : TIME := T#2S;
    uiRetryMax      : UINT := 2;
    tReconnectDelay : TIME := T#500MS;
    xUse4E          : BOOL := FALSE;
    xUseUdp         : BOOL := FALSE;
    uiSerialNo      : UINT := 1;
END_VAR
VAR_IN_OUT
    aWriteBits      : ARRAY[0..SLMP_MAX_BIT_INDEX] OF BOOL;
END_VAR
VAR_OUTPUT
    xBusy           : BOOL;
    xDone           : BOOL;
    xError          : BOOL;
    diError         : DINT;
    uiRetryCount    : UINT;
    aLastResponse   : ARRAY[0..SLMP_LAST_RESPONSE_INDEX_MAX] OF BYTE;
    uiLastResponseLen : UINT;
    uiLastEndCode   : UINT;
END_VAR
VAR
    fbWriteBit      : FB_SlmpWriteBitDevice;
    udInstanceId    : UDINT := 0;

    xExecPrev       : BOOL := FALSE;
    xPending        : BOOL := FALSE;
    xActive         : BOOL := FALSE;
    xExecPulse      : BOOL := FALSE;
    iLockIdx        : INT := -1;

    udiHeadLatched  : UDINT := 0;
    uiDeviceLatched : UINT := 0;
    uiPointsLatched : UINT := 0;
    uiSerialActive  : UINT := 0;
    aWriteLatched   : ARRAY[0..SLMP_MAX_BIT_INDEX] OF BOOL;

    idx             : UINT;
    uiSerialEff     : UINT;
    iSlot           : INT;
    iFreeSlot       : INT;
    xLocked         : BOOL;
END_VAR

// === IMPLEMENTATION ===
IF udInstanceId = 0 THEN
    GVL_SlmpRuntime.g_udServiceInstanceCounter := GVL_SlmpRuntime.g_udServiceInstanceCounter + 1;
    udInstanceId := GVL_SlmpRuntime.g_udServiceInstanceCounter;
    IF udInstanceId = 0 THEN
        udInstanceId := 1;
    END_IF;
END_IF;

IF xExecute AND (NOT xExecPrev) THEN
    IF (NOT xPending) AND (NOT xActive) THEN
        udiHeadLatched := udiHeadDevNo;
        uiDeviceLatched := uiDeviceCode;
        uiPointsLatched := uiPoints;
        FOR idx := 0 TO SLMP_MAX_BIT_INDEX DO
            aWriteLatched[idx] := aWriteBits[idx];
        END_FOR;
        xDone := FALSE;
        xError := FALSE;
        diError := 0;
        uiRetryCount := 0;
        xPending := TRUE;
    END_IF;
END_IF;
xExecPrev := xExecute;

xExecPulse := FALSE;
IF xPending AND (NOT xActive) THEN
    xLocked := FALSE;
    iFreeSlot := -1;
    FOR iSlot := 0 TO 7 DO
        IF (GVL_SlmpRuntime.g_aLockOwner[iSlot] <> 0) AND
           (GVL_SlmpRuntime.g_aLockIp[iSlot] = sIp) AND
           (GVL_SlmpRuntime.g_aLockPort[iSlot] = uiPort) AND
           (GVL_SlmpRuntime.g_aLockUseUdp[iSlot] = xUseUdp) THEN
            xLocked := TRUE;
            EXIT;
        END_IF;
        IF (iFreeSlot < 0) AND (GVL_SlmpRuntime.g_aLockOwner[iSlot] = 0) THEN
            iFreeSlot := iSlot;
        END_IF;
    END_FOR;

    IF (NOT xLocked) AND (iFreeSlot >= 0) THEN
        GVL_SlmpRuntime.g_aLockOwner[iFreeSlot] := udInstanceId;
        GVL_SlmpRuntime.g_aLockIp[iFreeSlot] := sIp;
        GVL_SlmpRuntime.g_aLockPort[iFreeSlot] := uiPort;
        GVL_SlmpRuntime.g_aLockUseUdp[iFreeSlot] := xUseUdp;
        iLockIdx := iFreeSlot;

        xActive := TRUE;
        xExecPulse := TRUE;
        IF xUse4E THEN
            uiSerialActive := F_SlmpNextSerialNo(uiSeed := uiSerialNo);
        END_IF;
    END_IF;
END_IF;

IF xActive THEN
    IF xUse4E THEN
        uiSerialEff := uiSerialActive;
        IF uiSerialEff = 0 THEN
            uiSerialEff := 1;
        END_IF;
    ELSE
        uiSerialEff := uiSerialNo;
    END_IF;

    fbWriteBit(
        xExecute := xExecPulse,
        sIp := sIp,
        uiPort := uiPort,
        udiHeadDevNo := udiHeadLatched,
        uiDeviceCode := uiDeviceLatched,
        xAutoSubCommand := TRUE,
        uiSubCommand := 0,
        uiPoints := uiPointsLatched,
        aWriteBits := aWriteLatched,
        tTimeout := tTimeout,
        uiRetryMax := uiRetryMax,
        tReconnectDelay := tReconnectDelay,
        xUse4E := xUse4E,
        xUseUdp := xUseUdp,
        uiSerialNo := uiSerialEff
    );
ELSE
    xBusy := xPending;
    IF NOT xExecute THEN
        xDone := FALSE;
        xError := FALSE;
        diError := 0;
        uiRetryCount := 0;
    END_IF;
    RETURN;
END_IF;

xBusy := fbWriteBit.xBusy;
xDone := fbWriteBit.xDone;
xError := fbWriteBit.xError;
diError := fbWriteBit.diError;
uiRetryCount := fbWriteBit.uiRetryCount;
FOR idx := 0 TO SLMP_LAST_RESPONSE_INDEX_MAX DO
    aLastResponse[idx] := fbWriteBit.aLastResponse[idx];
END_FOR;
uiLastResponseLen := fbWriteBit.uiLastResponseLen;
uiLastEndCode := fbWriteBit.uiLastEndCode;

IF fbWriteBit.xDone OR fbWriteBit.xError THEN
    xPending := FALSE;
    xActive := FALSE;
    IF iLockIdx >= 0 THEN
        GVL_SlmpRuntime.g_aLockOwner[iLockIdx] := 0;
        GVL_SlmpRuntime.g_aLockIp[iLockIdx] := '';
        GVL_SlmpRuntime.g_aLockPort[iLockIdx] := 0;
        GVL_SlmpRuntime.g_aLockUseUdp[iLockIdx] := FALSE;
        iLockIdx := -1;
    END_IF;
END_IF;

(* ---- FB_SlmpWriteDevice.st ---- *)
FUNCTION_BLOCK FB_SlmpWriteDevice
VAR_INPUT
    xExecute         : BOOL;
    sIp              : STRING;
    uiPort           : UINT;
    udiHeadDevNo     : UDINT := 100;
    uiDeviceCode     : UINT := 16#00A8; // D
    xAutoSubCommand  : BOOL := TRUE;
    uiSubCommand     : UINT := 16#0000; // 0000: word, 0001: bit
    uiPoints         : UINT := 1;
    aWriteBits       : ARRAY[0..SLMP_MAX_BIT_INDEX] OF BOOL;
    tTimeout         : TIME := T#2S;
    uiRetryMax       : UINT := 2;
    tReconnectDelay  : TIME := T#500MS;
    xUse4E           : BOOL := FALSE;
    uiSerialNo       : UINT := 0;
END_VAR
VAR_IN_OUT
    aWriteValues     : ARRAY[0..SLMP_MAX_WORD_INDEX] OF UINT;
END_VAR
VAR_OUTPUT
    xBusy            : BOOL;
    xDone            : BOOL;
    xError           : BOOL;
    diError          : DINT;
    uiRetryCount     : UINT;
    aLastResponse    : ARRAY[0..SLMP_LAST_RESPONSE_INDEX_MAX] OF BYTE;
    uiLastResponseLen: UINT;
    uiLastEndCode    : UINT;
END_VAR
VAR
    step             : INT := 0;
    xExecPrev        : BOOL := FALSE;

    fbCore           : FB_SlmpCore;

    tx               : ARRAY[0..SLMP_WRITE_TX_INDEX_MAX] OF BYTE;
    rx               : ARRAY[0..SLMP_LAST_RESPONSE_INDEX_MAX] OF BYTE;
    txLen            : LINT := 0;
    rxLen            : LINT := 0;
    lenReq           : UINT := 0;
    endCode          : UINT := 0;

    uiPointsReq      : UINT := 0;
    uiPointsEff      : UINT := 0;
    uiSubCmdEff      : UINT := 0;
    xBitMode         : BOOL := FALSE;
    idx              : UINT := 0;
    aWriteValuesLocal: ARRAY[0..SLMP_MAX_WORD_INDEX] OF UINT;
    iDataStart       : DINT := 21;
    iEndCodeStart    : DINT := 9;
    iMinRxLen        : LINT := 11;
    uiRxSerialNo     : UINT := 0;
    uiCopyLen        : UINT := 0;
    iPayloadBytes    : LINT := 0;
    iByteOffset      : DINT := 0;

    xStateTimeout    : BOOL := FALSE;
    xRetryTiming     : BOOL := FALSE;
    fbTimeout        : TON;
    fbReconnect      : TON;
END_VAR

// === IMPLEMENTATION ===
IF (xExecute AND NOT xExecPrev) THEN
    xBusy := TRUE;
    xDone := FALSE;
    xError := FALSE;
    diError := 0;
    uiRetryCount := 0;
    uiLastResponseLen := 0;
    uiLastEndCode := 0;
    FOR idx := 0 TO SLMP_LAST_RESPONSE_INDEX_MAX DO
        aLastResponse[idx] := 0;
    END_FOR;
    step := 10;
END_IF;
xExecPrev := xExecute;

xStateTimeout := (step = 20) OR (step = 40) OR (step = 50);
fbTimeout(IN := xStateTimeout, PT := tTimeout);
fbReconnect(IN := xRetryTiming, PT := tReconnectDelay);

IF (step <> 0) AND (step <> 80) AND fbTimeout.Q THEN
    diError := -2010;
    xError := TRUE;
    step := 90;
END_IF;

CASE step OF
    0:
        xRetryTiming := FALSE;

    10:
        uiSubCmdEff := F_SlmpResolveSubCommand(
            uiDeviceCode := uiDeviceCode,
            xAutoSubCommand := xAutoSubCommand,
            uiSubCommand := uiSubCommand
        );
        xBitMode := F_SlmpIsBitSubCommand(uiSubCommand := uiSubCmdEff);

        uiPointsReq := uiPoints;
        IF uiPointsReq = 0 THEN
            diError := -2000;
            xError := TRUE;
            xBusy := FALSE;
            step := 0;
        ELSE
            uiPointsEff := F_SlmpClampPoints(uiPoints := uiPointsReq, xBitMode := xBitMode);
        END_IF;

        IF NOT xBitMode THEN
            FOR idx := 0 TO SLMP_MAX_WORD_INDEX DO
                aWriteValuesLocal[idx] := aWriteValues[idx];
            END_FOR;
        END_IF;

        IF NOT xError THEN
            step := 20;
        END_IF;

    20:
        IF fbCore.OpenAndConnect(sIp := sIp, uiPort := uiPort) THEN
            step := 30;
        ELSE
            CASE fbCore.diLastError OF
                -1: diError := -2001;
                -2: diError := -2005;
                -3: diError := -2002;
            ELSE
                diError := -2002;
            END_CASE;
            xError := TRUE;
            step := 90;
        END_IF;

    30:
        IF xUse4E THEN
            iDataStart := 25;
            iEndCodeStart := 13;
            iMinRxLen := 15;
        ELSE
            iDataStart := 21;
            iEndCodeStart := 9;
            iMinRxLen := 11;
        END_IF;

        iPayloadBytes := BuildWritePayload();
        lenReq := TO_UINT(12 + TO_UINT(iPayloadBytes));

        IF xUse4E THEN
            tx[0] := 16#54; tx[1] := 16#00;
            tx[2] := TO_BYTE(uiSerialNo AND 16#00FF);
            tx[3] := TO_BYTE(SHR(uiSerialNo, 8) AND 16#00FF);
            tx[4] := 16#00; tx[5] := 16#00;
            tx[6] := 16#00;
            tx[7] := 16#FF;
            tx[8] := 16#FF; tx[9] := 16#03;
            tx[10] := 16#00;
            tx[11] := TO_BYTE(lenReq AND 16#00FF);
            tx[12] := TO_BYTE(SHR(lenReq, 8) AND 16#00FF);
            tx[13] := 16#10; tx[14] := 16#00;
            tx[15] := 16#01; tx[16] := 16#14;
            tx[17] := TO_BYTE(uiSubCmdEff AND 16#00FF);
            tx[18] := TO_BYTE(SHR(uiSubCmdEff, 8) AND 16#00FF);
            tx[19] := TO_BYTE(udiHeadDevNo AND 16#000000FF);
            tx[20] := TO_BYTE(SHR(udiHeadDevNo, 8) AND 16#000000FF);
            tx[21] := TO_BYTE(SHR(udiHeadDevNo, 16) AND 16#000000FF);
            tx[22] := TO_BYTE(uiDeviceCode AND 16#00FF);
            tx[23] := TO_BYTE(uiPointsEff AND 16#00FF);
            tx[24] := TO_BYTE(SHR(uiPointsEff, 8) AND 16#00FF);
        ELSE
            tx[0] := 16#50; tx[1] := 16#00;
            tx[2] := 16#00;
            tx[3] := 16#FF;
            tx[4] := 16#FF; tx[5] := 16#03;
            tx[6] := 16#00;
            tx[7] := TO_BYTE(lenReq AND 16#00FF);
            tx[8] := TO_BYTE(SHR(lenReq, 8) AND 16#00FF);
            tx[9] := 16#10; tx[10] := 16#00;
            tx[11] := 16#01; tx[12] := 16#14;
            tx[13] := TO_BYTE(uiSubCmdEff AND 16#00FF);
            tx[14] := TO_BYTE(SHR(uiSubCmdEff, 8) AND 16#00FF);
            tx[15] := TO_BYTE(udiHeadDevNo AND 16#000000FF);
            tx[16] := TO_BYTE(SHR(udiHeadDevNo, 8) AND 16#000000FF);
            tx[17] := TO_BYTE(SHR(udiHeadDevNo, 16) AND 16#000000FF);
            tx[18] := TO_BYTE(uiDeviceCode AND 16#00FF);
            tx[19] := TO_BYTE(uiPointsEff AND 16#00FF);
            tx[20] := TO_BYTE(SHR(uiPointsEff, 8) AND 16#00FF);
        END_IF;

        txLen := TO_LINT(iDataStart) + iPayloadBytes;
        step := 40;

    40:
        IF NOT fbCore.SendBytes(pData := ADR(tx[0]), liLen := txLen) THEN
            diError := -2003;
            xError := TRUE;
            step := 90;
        ELSE
            step := 50;
        END_IF;

    50:
        rxLen := fbCore.RecvBytes(pData := ADR(rx[0]), liMaxLen := SIZEOF(rx));
        IF rxLen > 0 THEN
            uiCopyLen := 0;
            IF rxLen > TO_LINT(SLMP_LAST_RESPONSE_INDEX_MAX + 1) THEN
                uiCopyLen := SLMP_LAST_RESPONSE_INDEX_MAX + 1;
            ELSE
                uiCopyLen := TO_UINT(rxLen);
            END_IF;
            uiLastResponseLen := uiCopyLen;
            IF uiCopyLen > 0 THEN
                FOR idx := 0 TO (uiCopyLen - 1) DO
                    aLastResponse[idx] := rx[idx];
                END_FOR;
            END_IF;
            IF rxLen < iMinRxLen THEN
                diError := -2004;
                xError := TRUE;
                step := 90;
            ELSE
                IF xUse4E THEN
                    uiRxSerialNo := TO_UINT(rx[2]) OR SHL(TO_UINT(rx[3]), 8);
                    IF uiRxSerialNo <> uiSerialNo THEN
                        // Drop stale frame and keep waiting until timeout.
                        rxLen := 0;
                        uiLastResponseLen := 0;
                    END_IF;
                END_IF;
            END_IF;
            IF (NOT xError) AND (rxLen > 0) THEN
                endCode := TO_UINT(rx[iEndCodeStart]) OR SHL(TO_UINT(rx[iEndCodeStart + 1]), 8);
                uiLastEndCode := endCode;
                IF endCode <> 0 THEN
                    diError := TO_DINT(endCode);
                    xError := TRUE;
                    step := 90;
                ELSE
                    xDone := TRUE;
                    xBusy := FALSE;
                    step := 90;
                END_IF;
            END_IF;
        END_IF;

    80:
        xRetryTiming := TRUE;
        IF fbReconnect.Q THEN
            xRetryTiming := FALSE;
            step := 10;
        END_IF;

    90:
        IF xError THEN
            fbCore.CloseSocket();
        END_IF;

        IF xError AND (uiRetryCount < uiRetryMax) THEN
            uiRetryCount := uiRetryCount + 1;
            xError := FALSE;
            step := 80;
        ELSE
            xBusy := FALSE;
            step := 0;
        END_IF;
END_CASE;
